// TwinCAT 3 PLC project PLC
// ProgramVersion: 3.1.4023.0
// libraries:
//   Tc2_Standard, * (Beckhoff Automation GmbH)
//   Tc2_System, * (Beckhoff Automation GmbH)
//   Tc3_Module, * (Beckhoff Automation GmbH)
// project tree:
//   / PlcTask.TcTTO
//   POUs/ MAIN.TcPOU
//   DUTs/IO/PdoEntries/ Status_E3F6A94B.TcDUT, Input_97D1F313.TcDUT, Status_B4798D86.TcDUT, Status_882A150F.TcDUT, Output_FFFF807A.TcDUT, Control_F189B737.TcDUT, Control_17BA1FC2.TcDUT
//   DUTs/IO/PDOs/ InfoData_6F19DB2B.TcDUT, Channel_42CA91F7.TcDUT, WcState_0B2B16F9.TcDUT, AI_Inputs_5AF6604E.TcDUT, WcState_9091E0EB.TcDUT, InfoData_32EB74EA.TcDUT, AI_Input_Channel_5AF6604E.TcDUT, Digital_BD004D6F.TcDUT, Encoder_Channel_2E4EA213.TcDUT, Digital_A7E1DFAB.TcDUT, Analog_Channel_5F9B7EA6.TcDUT, Encoder_Channel_B7999E14.TcDUT, DI_Inputs_BD004D6F.TcDUT, ENC_Inputs_Channel_69C51E8E.TcDUT, PLS_Inputs_5A35B63D.TcDUT, DO_Outputs_A7E1DFAB.TcDUT, AO_Output_Channel_BA7EBB7C.TcDUT, ENC_Outputs_Channel_DC4E290B.TcDUT, PLS_Outputs_AFB7DAF5.TcDUT, ENC_Inputs_Channel_6B6F9807.TcDUT, DI_Inputs_9882B618.TcDUT, ENC_Inputs_Channel_E5B5E929.TcDUT, PLS_Inputs_65C9A3D6.TcDUT, DO_Outputs_47E26D6A.TcDUT, ENC_Outputs_Channel_2E82BC43.TcDUT, PLS_Outputs_8EABC224.TcDUT, InfoData_E68C61CD.TcDUT, InfoData_2A97D6CF.TcDUT, Inputs_25A0042B.TcDUT, Outputs_2397A10E.TcDUT
//   DUTs/IO/Boxes/ EK1100_1FC0878B.TcDUT, EK1122_1FC0878B.TcDUT, EM2042_2B6483BD.TcDUT, EM3701_AB0D469D.TcDUT, EM3702_FDD84FD8.TcDUT, EM3712_FDD84FD8.TcDUT, EM7004_866015E1.TcDUT, EM7004_7586CC95.TcDUT, EM7004_5FA1DD22.TcDUT, EM7004_0F97553F.TcDUT
//   DUTs/IO/Devices/ SyncUnitTask_2D604ED5.TcDUT, SyncUnitTasks_6FEB8257.TcDUT, SyncUnits_99E584AF.TcDUT
//   DUTs/IO/Topology/ Beckhoff_EM2xxxEK1122_B7C04D41.TcDUT, Beckhoff_EM2xxx_23EB33C6.TcDUT, Beckhoff_EM3xxxEK1122_FEF78CCD.TcDUT, Beckhoff_EM3xxx_ABA31799.TcDUT, Beckhoff_EM7xxxEK1122_DEE9974A.TcDUT, Beckhoff_EM7xxx_9745B8AE.TcDUT, EtherCAT_Master_EMxxxx_E69B3047.TcDUT
//   DUTs/IO/Base/ EtcSlaveBase_82538BE2.TcDUT, EtcSlaveBase_82538BE2.TcDUT, EtcSlaveBase_82538BE2.TcDUT, EtcSlaveTerminalBase_947E5A46.TcDUT, EtcSlaveBoxBase_77A0E4A7.TcDUT, EtcSlaveEndTerminalBase_866C7F0C.TcDUT, InputBase_8311D824.TcDUT, OutputBase_10CEE7DE.TcDUT, EtcMasterBase_62654B43.TcDUT
//   GVLs/ GVL_iXlinker.TcGVL
// real-time tasks:
//   TASK PlcTask: cycle T#10ms, priority 20, ADS port 350
// I/O:
//   DEVICE EtherCAT_Master_EMxxxx, AmsNetId 172.20.30.238.12.1
//     Beckhoff EM2xxx [EK1100 EtherCAT Coupler (2A E-Bus)]
//       Beckhoff EM2xxxEK1122 [EK1122 2 port EtherCAT junction]
//         Beckhoff EM2xxxsub EK1100 [EK1100 EtherCAT Coupler (2A E-Bus)]
//       A_0001(EM2042-0000-0016) [EM2042 16Ch. Dig. Output 24V, 0.5A, D-Sub connection]
//       A_0002(EM2042-0000-0017) [EM2042 16Ch. Dig. Output 24V, 0.5A, D-Sub connection]
//     Beckhoff EM3xxx [EK1100 EtherCAT Coupler (2A E-Bus)]
//       Beckhoff EM3xxxEK1122 [EK1122 2 port EtherCAT junction]
//         Beckhoff EM3xxxsub EK1100 [EK1100 EtherCAT Coupler (2A E-Bus)]
//       A_0001(EM3701-0000-0016) [EM3701, 1Ch. differential pressure measuring terminal 100hPa (100mbar)]
//       A_0002(EM3702-0000-0016) [EM3702  2Ch. relative pressure measuring terminal 7,500 hPa (7.5 bar)]
//       A_0003(EM3712-0000-0016) [EM3712  2Ch relative pressure measuring terminal -1,000...+1,000 hPa (-1...+1 bar)]
//     Beckhoff EM7xxx [EK1100 EtherCAT Coupler (2A E-Bus)]
//       Beckhoff EM7xxxEK1122 [EK1122 2 port EtherCAT junction]
//         Beckhoff EM7xxxsub EK1100 [EK1100 EtherCAT Coupler (2A E-Bus)]
//       A_0001(EM7004-0000-9995) [EM7004 4-Axis Interface Unit]
//       A_0002(EM7004-0000-9996) [EM7004 4-Axis Interface Unit]
//       A_0003(EM7004-0000-9997) [EM7004 4-Axis Interface Unit]
//       A_0004(EM7004-0000-0016) [EM7004 4-Axis Interface Unit]
//       A_0005(EM7004-0000-0017) [EM7004 4-Axis Interface Unit]
//       A_0006(EM7004-0000-0018) [EM7004 4-Axis Interface Unit]
// variable links:
//   PLC/PLC Instance <-> EtherCAT Master EMxxxx/Beckhoff EM2xxx
//     PlcTask Inputs/GVL_iXlinker.EtherCAT_Master_EMxxxx.Beckhoff_EM2xxx.InfoData.State <-> InfoData/State
//   PLC/PLC Instance <-> EtherCAT Master EMxxxx/Beckhoff EM2xxx/Beckhoff EM2xxxEK1122
//     PlcTask Inputs/GVL_iXlinker.EtherCAT_Master_EMxxxx.Beckhoff_EM2xxx.Beckhoff_EM2xxxEK1122.InfoData.State <-> InfoData/State
//   PLC/PLC Instance <-> EtherCAT Master EMxxxx/Beckhoff EM2xxx/Beckhoff EM2xxxEK1122/Beckhoff EM2xxxsub EK1100
//     PlcTask Inputs/GVL_iXlinker.EtherCAT_Master_EMxxxx.Beckhoff_EM2xxx.Beckhoff_EM2xxxEK1122.Beckhoff_EM2xxxsub_EK1100.InfoData.State <-> InfoData/State
//   PLC/PLC Instance <-> EtherCAT Master EMxxxx/Beckhoff EM2xxx/A_0001(EM2042-0000-0016)
//     PlcTask Outputs/GVL_iXlinker.EtherCAT_Master_EMxxxx.Beckhoff_EM2xxx.A_0001_EM2042_0000_0016.Channel_1.Output <-> Channel 1/Output
//     PlcTask Outputs/GVL_iXlinker.EtherCAT_Master_EMxxxx.Beckhoff_EM2xxx.A_0001_EM2042_0000_0016.Channel_2.Output <-> Channel 2/Output
//     PlcTask Outputs/GVL_iXlinker.EtherCAT_Master_EMxxxx.Beckhoff_EM2xxx.A_0001_EM2042_0000_0016.Channel_3.Output <-> Channel 3/Output
//     PlcTask Outputs/GVL_iXlinker.EtherCAT_Master_EMxxxx.Beckhoff_EM2xxx.A_0001_EM2042_0000_0016.Channel_4.Output <-> Channel 4/Output
//     PlcTask Outputs/GVL_iXlinker.EtherCAT_Master_EMxxxx.Beckhoff_EM2xxx.A_0001_EM2042_0000_0016.Channel_5.Output <-> Channel 5/Output
//     PlcTask Outputs/GVL_iXlinker.EtherCAT_Master_EMxxxx.Beckhoff_EM2xxx.A_0001_EM2042_0000_0016.Channel_6.Output <-> Channel 6/Output
//     PlcTask Outputs/GVL_iXlinker.EtherCAT_Master_EMxxxx.Beckhoff_EM2xxx.A_0001_EM2042_0000_0016.Channel_7.Output <-> Channel 7/Output
//     PlcTask Outputs/GVL_iXlinker.EtherCAT_Master_EMxxxx.Beckhoff_EM2xxx.A_0001_EM2042_0000_0016.Channel_8.Output <-> Channel 8/Output
//     PlcTask Outputs/GVL_iXlinker.EtherCAT_Master_EMxxxx.Beckhoff_EM2xxx.A_0001_EM2042_0000_0016.Channel_9.Output <-> Channel 9/Output
//     PlcTask Outputs/GVL_iXlinker.EtherCAT_Master_EMxxxx.Beckhoff_EM2xxx.A_0001_EM2042_0000_0016.Channel_10.Output <-> Channel 10/Output
//     PlcTask Outputs/GVL_iXlinker.EtherCAT_Master_EMxxxx.Beckhoff_EM2xxx.A_0001_EM2042_0000_0016.Channel_11.Output <-> Channel 11/Output
//     PlcTask Outputs/GVL_iXlinker.EtherCAT_Master_EMxxxx.Beckhoff_EM2xxx.A_0001_EM2042_0000_0016.Channel_12.Output <-> Channel 12/Output
//     PlcTask Outputs/GVL_iXlinker.EtherCAT_Master_EMxxxx.Beckhoff_EM2xxx.A_0001_EM2042_0000_0016.Channel_13.Output <-> Channel 13/Output
//     PlcTask Outputs/GVL_iXlinker.EtherCAT_Master_EMxxxx.Beckhoff_EM2xxx.A_0001_EM2042_0000_0016.Channel_14.Output <-> Channel 14/Output
//     PlcTask Outputs/GVL_iXlinker.EtherCAT_Master_EMxxxx.Beckhoff_EM2xxx.A_0001_EM2042_0000_0016.Channel_15.Output <-> Channel 15/Output
//     PlcTask Outputs/GVL_iXlinker.EtherCAT_Master_EMxxxx.Beckhoff_EM2xxx.A_0001_EM2042_0000_0016.Channel_16.Output <-> Channel 16/Output
//     PlcTask Inputs/GVL_iXlinker.EtherCAT_Master_EMxxxx.Beckhoff_EM2xxx.A_0001_EM2042_0000_0016.WcState.WcState <-> WcState/WcState
//     PlcTask Inputs/GVL_iXlinker.EtherCAT_Master_EMxxxx.Beckhoff_EM2xxx.A_0001_EM2042_0000_0016.InfoData.State <-> InfoData/State
//   PLC/PLC Instance <-> EtherCAT Master EMxxxx/Beckhoff EM2xxx/A_0002(EM2042-0000-0017)
//     PlcTask Outputs/GVL_iXlinker.EtherCAT_Master_EMxxxx.Beckhoff_EM2xxx.A_0002_EM2042_0000_0017.Channel_1.Output <-> Channel 1/Output
//     PlcTask Outputs/GVL_iXlinker.EtherCAT_Master_EMxxxx.Beckhoff_EM2xxx.A_0002_EM2042_0000_0017.Channel_2.Output <-> Channel 2/Output
//     PlcTask Outputs/GVL_iXlinker.EtherCAT_Master_EMxxxx.Beckhoff_EM2xxx.A_0002_EM2042_0000_0017.Channel_3.Output <-> Channel 3/Output
//     PlcTask Outputs/GVL_iXlinker.EtherCAT_Master_EMxxxx.Beckhoff_EM2xxx.A_0002_EM2042_0000_0017.Channel_4.Output <-> Channel 4/Output
//     PlcTask Outputs/GVL_iXlinker.EtherCAT_Master_EMxxxx.Beckhoff_EM2xxx.A_0002_EM2042_0000_0017.Channel_5.Output <-> Channel 5/Output
//     PlcTask Outputs/GVL_iXlinker.EtherCAT_Master_EMxxxx.Beckhoff_EM2xxx.A_0002_EM2042_0000_0017.Channel_6.Output <-> Channel 6/Output
//     PlcTask Outputs/GVL_iXlinker.EtherCAT_Master_EMxxxx.Beckhoff_EM2xxx.A_0002_EM2042_0000_0017.Channel_7.Output <-> Channel 7/Output
//     PlcTask Outputs/GVL_iXlinker.EtherCAT_Master_EMxxxx.Beckhoff_EM2xxx.A_0002_EM2042_0000_0017.Channel_8.Output <-> Channel 8/Output
//     PlcTask Outputs/GVL_iXlinker.EtherCAT_Master_EMxxxx.Beckhoff_EM2xxx.A_0002_EM2042_0000_0017.Channel_9.Output <-> Channel 9/Output
//     PlcTask Outputs/GVL_iXlinker.EtherCAT_Master_EMxxxx.Beckhoff_EM2xxx.A_0002_EM2042_0000_0017.Channel_10.Output <-> Channel 10/Output
//     PlcTask Outputs/GVL_iXlinker.EtherCAT_Master_EMxxxx.Beckhoff_EM2xxx.A_0002_EM2042_0000_0017.Channel_11.Output <-> Channel 11/Output
//     PlcTask Outputs/GVL_iXlinker.EtherCAT_Master_EMxxxx.Beckhoff_EM2xxx.A_0002_EM2042_0000_0017.Channel_12.Output <-> Channel 12/Output
//     PlcTask Outputs/GVL_iXlinker.EtherCAT_Master_EMxxxx.Beckhoff_EM2xxx.A_0002_EM2042_0000_0017.Channel_13.Output <-> Channel 13/Output
//     PlcTask Outputs/GVL_iXlinker.EtherCAT_Master_EMxxxx.Beckhoff_EM2xxx.A_0002_EM2042_0000_0017.Channel_14.Output <-> Channel 14/Output
//     PlcTask Outputs/GVL_iXlinker.EtherCAT_Master_EMxxxx.Beckhoff_EM2xxx.A_0002_EM2042_0000_0017.Channel_15.Output <-> Channel 15/Output
//     PlcTask Outputs/GVL_iXlinker.EtherCAT_Master_EMxxxx.Beckhoff_EM2xxx.A_0002_EM2042_0000_0017.Channel_16.Output <-> Channel 16/Output
//     PlcTask Inputs/GVL_iXlinker.EtherCAT_Master_EMxxxx.Beckhoff_EM2xxx.A_0002_EM2042_0000_0017.WcState.WcState <-> WcState/WcState
//     PlcTask Inputs/GVL_iXlinker.EtherCAT_Master_EMxxxx.Beckhoff_EM2xxx.A_0002_EM2042_0000_0017.InfoData.State <-> InfoData/State
//   PLC/PLC Instance <-> EtherCAT Master EMxxxx/Beckhoff EM3xxx
//     PlcTask Inputs/GVL_iXlinker.EtherCAT_Master_EMxxxx.Beckhoff_EM3xxx.InfoData.State <-> InfoData/State
//   PLC/PLC Instance <-> EtherCAT Master EMxxxx/Beckhoff EM3xxx/Beckhoff EM3xxxEK1122
//     PlcTask Inputs/GVL_iXlinker.EtherCAT_Master_EMxxxx.Beckhoff_EM3xxx.Beckhoff_EM3xxxEK1122.InfoData.State <-> InfoData/State
//   PLC/PLC Instance <-> EtherCAT Master EMxxxx/Beckhoff EM3xxx/Beckhoff EM3xxxEK1122/Beckhoff EM3xxxsub EK1100
//     PlcTask Inputs/GVL_iXlinker.EtherCAT_Master_EMxxxx.Beckhoff_EM3xxx.Beckhoff_EM3xxxEK1122.Beckhoff_EM3xxxsub_EK1100.InfoData.State <-> InfoData/State
//   PLC/PLC Instance <-> EtherCAT Master EMxxxx/Beckhoff EM3xxx/A_0001(EM3701-0000-0016)
//     PlcTask Inputs/GVL_iXlinker.EtherCAT_Master_EMxxxx.Beckhoff_EM3xxx.A_0001_EM3701_0000_0016.AI_Inputs.Status/Underrange <-> AI Inputs/Status/Underrange
//     PlcTask Inputs/GVL_iXlinker.EtherCAT_Master_EMxxxx.Beckhoff_EM3xxx.A_0001_EM3701_0000_0016.AI_Inputs.Status/Overrange <-> AI Inputs/Status/Overrange
//     PlcTask Inputs/GVL_iXlinker.EtherCAT_Master_EMxxxx.Beckhoff_EM3xxx.A_0001_EM3701_0000_0016.AI_Inputs.Status/Limit_1 <-> AI Inputs/Status/Limit 1
//     PlcTask Inputs/GVL_iXlinker.EtherCAT_Master_EMxxxx.Beckhoff_EM3xxx.A_0001_EM3701_0000_0016.AI_Inputs.Status/Limit_2 <-> AI Inputs/Status/Limit 2
//     PlcTask Inputs/GVL_iXlinker.EtherCAT_Master_EMxxxx.Beckhoff_EM3xxx.A_0001_EM3701_0000_0016.AI_Inputs.Status/Error <-> AI Inputs/Status/Error
//     PlcTask Inputs/GVL_iXlinker.EtherCAT_Master_EMxxxx.Beckhoff_EM3xxx.A_0001_EM3701_0000_0016.AI_Inputs.Status/TxPDO_State <-> AI Inputs/Status/TxPDO State
//     PlcTask Inputs/GVL_iXlinker.EtherCAT_Master_EMxxxx.Beckhoff_EM3xxx.A_0001_EM3701_0000_0016.AI_Inputs.Value <-> AI Inputs/Value
//     PlcTask Inputs/GVL_iXlinker.EtherCAT_Master_EMxxxx.Beckhoff_EM3xxx.A_0001_EM3701_0000_0016.WcState.WcState <-> WcState/WcState
//     PlcTask Inputs/GVL_iXlinker.EtherCAT_Master_EMxxxx.Beckhoff_EM3xxx.A_0001_EM3701_0000_0016.WcState.InputToggle <-> WcState/InputToggle
//     PlcTask Inputs/GVL_iXlinker.EtherCAT_Master_EMxxxx.Beckhoff_EM3xxx.A_0001_EM3701_0000_0016.InfoData.AdsAddr <-> InfoData/AdsAddr
//     PlcTask Inputs/GVL_iXlinker.EtherCAT_Master_EMxxxx.Beckhoff_EM3xxx.A_0001_EM3701_0000_0016.InfoData.State <-> InfoData/State
//   PLC/PLC Instance <-> EtherCAT Master EMxxxx/Beckhoff EM3xxx/A_0002(EM3702-0000-0016)
//     PlcTask Inputs/GVL_iXlinker.EtherCAT_Master_EMxxxx.Beckhoff_EM3xxx.A_0002_EM3702_0000_0016.AI_Input_Channel_1.Status/Underrange <-> AI Input Channel 1/Status/Underrange
//     PlcTask Inputs/GVL_iXlinker.EtherCAT_Master_EMxxxx.Beckhoff_EM3xxx.A_0002_EM3702_0000_0016.AI_Input_Channel_2.Status/Underrange <-> AI Input Channel 2/Status/Underrange
//     PlcTask Inputs/GVL_iXlinker.EtherCAT_Master_EMxxxx.Beckhoff_EM3xxx.A_0002_EM3702_0000_0016.AI_Input_Channel_1.Status/Overrange <-> AI Input Channel 1/Status/Overrange
//     PlcTask Inputs/GVL_iXlinker.EtherCAT_Master_EMxxxx.Beckhoff_EM3xxx.A_0002_EM3702_0000_0016.AI_Input_Channel_2.Status/Overrange <-> AI Input Channel 2/Status/Overrange
//     PlcTask Inputs/GVL_iXlinker.EtherCAT_Master_EMxxxx.Beckhoff_EM3xxx.A_0002_EM3702_0000_0016.AI_Input_Channel_1.Status/Limit_1 <-> AI Input Channel 1/Status/Limit 1
//     PlcTask Inputs/GVL_iXlinker.EtherCAT_Master_EMxxxx.Beckhoff_EM3xxx.A_0002_EM3702_0000_0016.AI_Input_Channel_1.Status/Limit_2 <-> AI Input Channel 1/Status/Limit 2
//     PlcTask Inputs/GVL_iXlinker.EtherCAT_Master_EMxxxx.Beckhoff_EM3xxx.A_0002_EM3702_0000_0016.AI_Input_Channel_2.Status/Limit_1 <-> AI Input Channel 2/Status/Limit 1
//     PlcTask Inputs/GVL_iXlinker.EtherCAT_Master_EMxxxx.Beckhoff_EM3xxx.A_0002_EM3702_0000_0016.AI_Input_Channel_2.Status/Limit_2 <-> AI Input Channel 2/Status/Limit 2
//     PlcTask Inputs/GVL_iXlinker.EtherCAT_Master_EMxxxx.Beckhoff_EM3xxx.A_0002_EM3702_0000_0016.AI_Input_Channel_1.Status/Error <-> AI Input Channel 1/Status/Error
//     PlcTask Inputs/GVL_iXlinker.EtherCAT_Master_EMxxxx.Beckhoff_EM3xxx.A_0002_EM3702_0000_0016.AI_Input_Channel_2.Status/Error <-> AI Input Channel 2/Status/Error
//     PlcTask Inputs/GVL_iXlinker.EtherCAT_Master_EMxxxx.Beckhoff_EM3xxx.A_0002_EM3702_0000_0016.AI_Input_Channel_1.Status/TxPDO_State <-> AI Input Channel 1/Status/TxPDO State
//     PlcTask Inputs/GVL_iXlinker.EtherCAT_Master_EMxxxx.Beckhoff_EM3xxx.A_0002_EM3702_0000_0016.AI_Input_Channel_2.Status/TxPDO_State <-> AI Input Channel 2/Status/TxPDO State
//     PlcTask Inputs/GVL_iXlinker.EtherCAT_Master_EMxxxx.Beckhoff_EM3xxx.A_0002_EM3702_0000_0016.AI_Input_Channel_1.Value <-> AI Input Channel 1/Value
//     PlcTask Inputs/GVL_iXlinker.EtherCAT_Master_EMxxxx.Beckhoff_EM3xxx.A_0002_EM3702_0000_0016.AI_Input_Channel_2.Value <-> AI Input Channel 2/Value
//     PlcTask Inputs/GVL_iXlinker.EtherCAT_Master_EMxxxx.Beckhoff_EM3xxx.A_0002_EM3702_0000_0016.WcState.WcState <-> WcState/WcState
//     PlcTask Inputs/GVL_iXlinker.EtherCAT_Master_EMxxxx.Beckhoff_EM3xxx.A_0002_EM3702_0000_0016.WcState.InputToggle <-> WcState/InputToggle
//     PlcTask Inputs/GVL_iXlinker.EtherCAT_Master_EMxxxx.Beckhoff_EM3xxx.A_0002_EM3702_0000_0016.InfoData.AdsAddr <-> InfoData/AdsAddr
//     PlcTask Inputs/GVL_iXlinker.EtherCAT_Master_EMxxxx.Beckhoff_EM3xxx.A_0002_EM3702_0000_0016.InfoData.State <-> InfoData/State
//   PLC/PLC Instance <-> EtherCAT Master EMxxxx/Beckhoff EM3xxx/A_0003(EM3712-0000-0016)
//     PlcTask Inputs/GVL_iXlinker.EtherCAT_Master_EMxxxx.Beckhoff_EM3xxx.A_0003_EM3712_0000_0016.AI_Input_Channel_1.Status/Underrange <-> AI Input Channel 1/Status/Underrange
//     PlcTask Inputs/GVL_iXlinker.EtherCAT_Master_EMxxxx.Beckhoff_EM3xxx.A_0003_EM3712_0000_0016.AI_Input_Channel_2.Status/Underrange <-> AI Input Channel 2/Status/Underrange
//     PlcTask Inputs/GVL_iXlinker.EtherCAT_Master_EMxxxx.Beckhoff_EM3xxx.A_0003_EM3712_0000_0016.AI_Input_Channel_1.Status/Overrange <-> AI Input Channel 1/Status/Overrange
//     PlcTask Inputs/GVL_iXlinker.EtherCAT_Master_EMxxxx.Beckhoff_EM3xxx.A_0003_EM3712_0000_0016.AI_Input_Channel_2.Status/Overrange <-> AI Input Channel 2/Status/Overrange
//     PlcTask Inputs/GVL_iXlinker.EtherCAT_Master_EMxxxx.Beckhoff_EM3xxx.A_0003_EM3712_0000_0016.AI_Input_Channel_1.Status/Limit_1 <-> AI Input Channel 1/Status/Limit 1
//     PlcTask Inputs/GVL_iXlinker.EtherCAT_Master_EMxxxx.Beckhoff_EM3xxx.A_0003_EM3712_0000_0016.AI_Input_Channel_1.Status/Limit_2 <-> AI Input Channel 1/Status/Limit 2
//     PlcTask Inputs/GVL_iXlinker.EtherCAT_Master_EMxxxx.Beckhoff_EM3xxx.A_0003_EM3712_0000_0016.AI_Input_Channel_2.Status/Limit_1 <-> AI Input Channel 2/Status/Limit 1
//     PlcTask Inputs/GVL_iXlinker.EtherCAT_Master_EMxxxx.Beckhoff_EM3xxx.A_0003_EM3712_0000_0016.AI_Input_Channel_2.Status/Limit_2 <-> AI Input Channel 2/Status/Limit 2
//     PlcTask Inputs/GVL_iXlinker.EtherCAT_Master_EMxxxx.Beckhoff_EM3xxx.A_0003_EM3712_0000_0016.AI_Input_Channel_1.Status/Error <-> AI Input Channel 1/Status/Error
//     PlcTask Inputs/GVL_iXlinker.EtherCAT_Master_EMxxxx.Beckhoff_EM3xxx.A_0003_EM3712_0000_0016.AI_Input_Channel_2.Status/Error <-> AI Input Channel 2/Status/Error
//     PlcTask Inputs/GVL_iXlinker.EtherCAT_Master_EMxxxx.Beckhoff_EM3xxx.A_0003_EM3712_0000_0016.AI_Input_Channel_1.Status/TxPDO_State <-> AI Input Channel 1/Status/TxPDO State
//     PlcTask Inputs/GVL_iXlinker.EtherCAT_Master_EMxxxx.Beckhoff_EM3xxx.A_0003_EM3712_0000_0016.AI_Input_Channel_2.Status/TxPDO_State <-> AI Input Channel 2/Status/TxPDO State
//     PlcTask Inputs/GVL_iXlinker.EtherCAT_Master_EMxxxx.Beckhoff_EM3xxx.A_0003_EM3712_0000_0016.AI_Input_Channel_1.Value <-> AI Input Channel 1/Value
//     PlcTask Inputs/GVL_iXlinker.EtherCAT_Master_EMxxxx.Beckhoff_EM3xxx.A_0003_EM3712_0000_0016.AI_Input_Channel_2.Value <-> AI Input Channel 2/Value
//     PlcTask Inputs/GVL_iXlinker.EtherCAT_Master_EMxxxx.Beckhoff_EM3xxx.A_0003_EM3712_0000_0016.WcState.WcState <-> WcState/WcState
//     PlcTask Inputs/GVL_iXlinker.EtherCAT_Master_EMxxxx.Beckhoff_EM3xxx.A_0003_EM3712_0000_0016.WcState.InputToggle <-> WcState/InputToggle
//     PlcTask Inputs/GVL_iXlinker.EtherCAT_Master_EMxxxx.Beckhoff_EM3xxx.A_0003_EM3712_0000_0016.InfoData.AdsAddr <-> InfoData/AdsAddr
//     PlcTask Inputs/GVL_iXlinker.EtherCAT_Master_EMxxxx.Beckhoff_EM3xxx.A_0003_EM3712_0000_0016.InfoData.State <-> InfoData/State
//   PLC/PLC Instance <-> EtherCAT Master EMxxxx/Beckhoff EM7xxx
//     PlcTask Inputs/GVL_iXlinker.EtherCAT_Master_EMxxxx.Beckhoff_EM7xxx.InfoData.State <-> InfoData/State
//   PLC/PLC Instance <-> EtherCAT Master EMxxxx/Beckhoff EM7xxx/Beckhoff EM7xxxEK1122
//     PlcTask Inputs/GVL_iXlinker.EtherCAT_Master_EMxxxx.Beckhoff_EM7xxx.Beckhoff_EM7xxxEK1122.InfoData.State <-> InfoData/State
//   PLC/PLC Instance <-> EtherCAT Master EMxxxx/Beckhoff EM7xxx/Beckhoff EM7xxxEK1122/Beckhoff EM7xxxsub EK1100
//     PlcTask Inputs/GVL_iXlinker.EtherCAT_Master_EMxxxx.Beckhoff_EM7xxx.Beckhoff_EM7xxxEK1122.Beckhoff_EM7xxxsub_EK1100.InfoData.State <-> InfoData/State
//   PLC/PLC Instance <-> EtherCAT Master EMxxxx/Beckhoff EM7xxx/A_0001(EM7004-0000-9995)
//     PlcTask Inputs/GVL_iXlinker.EtherCAT_Master_EMxxxx.Beckhoff_EM7xxx.A_0001_EM7004_0000_9995.Digital.Input[0] <-> Digital/Input 0
//     PlcTask Inputs/GVL_iXlinker.EtherCAT_Master_EMxxxx.Beckhoff_EM7xxx.A_0001_EM7004_0000_9995.Digital.Input[1] <-> Digital/Input 1
//     PlcTask Inputs/GVL_iXlinker.EtherCAT_Master_EMxxxx.Beckhoff_EM7xxx.A_0001_EM7004_0000_9995.Digital.Input[2] <-> Digital/Input 2
//     PlcTask Inputs/GVL_iXlinker.EtherCAT_Master_EMxxxx.Beckhoff_EM7xxx.A_0001_EM7004_0000_9995.Digital.Input[3] <-> Digital/Input 3
//     PlcTask Inputs/GVL_iXlinker.EtherCAT_Master_EMxxxx.Beckhoff_EM7xxx.A_0001_EM7004_0000_9995.Digital.Input[4] <-> Digital/Input 4
//     PlcTask Inputs/GVL_iXlinker.EtherCAT_Master_EMxxxx.Beckhoff_EM7xxx.A_0001_EM7004_0000_9995.Digital.Input[5] <-> Digital/Input 5
//     PlcTask Inputs/GVL_iXlinker.EtherCAT_Master_EMxxxx.Beckhoff_EM7xxx.A_0001_EM7004_0000_9995.Digital.Input[6] <-> Digital/Input 6
//     PlcTask Inputs/GVL_iXlinker.EtherCAT_Master_EMxxxx.Beckhoff_EM7xxx.A_0001_EM7004_0000_9995.Digital.Input[7] <-> Digital/Input 7
//     PlcTask Inputs/GVL_iXlinker.EtherCAT_Master_EMxxxx.Beckhoff_EM7xxx.A_0001_EM7004_0000_9995.Digital.Input[8] <-> Digital/Input 8
//     PlcTask Inputs/GVL_iXlinker.EtherCAT_Master_EMxxxx.Beckhoff_EM7xxx.A_0001_EM7004_0000_9995.Digital.Input[9] <-> Digital/Input 9
//     PlcTask Inputs/GVL_iXlinker.EtherCAT_Master_EMxxxx.Beckhoff_EM7xxx.A_0001_EM7004_0000_9995.Digital.Input[10] <-> Digital/Input 10
//     PlcTask Inputs/GVL_iXlinker.EtherCAT_Master_EMxxxx.Beckhoff_EM7xxx.A_0001_EM7004_0000_9995.Digital.Input[11] <-> Digital/Input 11
//     PlcTask Inputs/GVL_iXlinker.EtherCAT_Master_EMxxxx.Beckhoff_EM7xxx.A_0001_EM7004_0000_9995.Digital.Input[12] <-> Digital/Input 12
//     PlcTask Inputs/GVL_iXlinker.EtherCAT_Master_EMxxxx.Beckhoff_EM7xxx.A_0001_EM7004_0000_9995.Digital.Input[13] <-> Digital/Input 13
//     PlcTask Inputs/GVL_iXlinker.EtherCAT_Master_EMxxxx.Beckhoff_EM7xxx.A_0001_EM7004_0000_9995.Digital.Input[14] <-> Digital/Input 14
//     PlcTask Inputs/GVL_iXlinker.EtherCAT_Master_EMxxxx.Beckhoff_EM7xxx.A_0001_EM7004_0000_9995.Digital.Input[15] <-> Digital/Input 15
//     PlcTask Inputs/GVL_iXlinker.EtherCAT_Master_EMxxxx.Beckhoff_EM7xxx.A_0001_EM7004_0000_9995.Encoder_Channel_1.Status <-> Encoder, Channel 1/Status
//     PlcTask Inputs/GVL_iXlinker.EtherCAT_Master_EMxxxx.Beckhoff_EM7xxx.A_0001_EM7004_0000_9995.Encoder_Channel_2.Status <-> Encoder, Channel 2/Status
//     PlcTask Inputs/GVL_iXlinker.EtherCAT_Master_EMxxxx.Beckhoff_EM7xxx.A_0001_EM7004_0000_9995.Encoder_Channel_3.Status <-> Encoder, Channel 3/Status
//     PlcTask Inputs/GVL_iXlinker.EtherCAT_Master_EMxxxx.Beckhoff_EM7xxx.A_0001_EM7004_0000_9995.Encoder_Channel_4.Status <-> Encoder, Channel 4/Status
//     PlcTask Inputs/GVL_iXlinker.EtherCAT_Master_EMxxxx.Beckhoff_EM7xxx.A_0001_EM7004_0000_9995.Encoder_Channel_1.Value <-> Encoder, Channel 1/Value
//     PlcTask Inputs/GVL_iXlinker.EtherCAT_Master_EMxxxx.Beckhoff_EM7xxx.A_0001_EM7004_0000_9995.Encoder_Channel_2.Value <-> Encoder, Channel 2/Value
//     PlcTask Inputs/GVL_iXlinker.EtherCAT_Master_EMxxxx.Beckhoff_EM7xxx.A_0001_EM7004_0000_9995.Encoder_Channel_3.Value <-> Encoder, Channel 3/Value
//     PlcTask Inputs/GVL_iXlinker.EtherCAT_Master_EMxxxx.Beckhoff_EM7xxx.A_0001_EM7004_0000_9995.Encoder_Channel_4.Value <-> Encoder, Channel 4/Value
//     PlcTask Inputs/GVL_iXlinker.EtherCAT_Master_EMxxxx.Beckhoff_EM7xxx.A_0001_EM7004_0000_9995.Encoder_Channel_1.Latch <-> Encoder, Channel 1/Latch
//     PlcTask Inputs/GVL_iXlinker.EtherCAT_Master_EMxxxx.Beckhoff_EM7xxx.A_0001_EM7004_0000_9995.Encoder_Channel_2.Latch <-> Encoder, Channel 2/Latch
//     PlcTask Inputs/GVL_iXlinker.EtherCAT_Master_EMxxxx.Beckhoff_EM7xxx.A_0001_EM7004_0000_9995.Encoder_Channel_3.Latch <-> Encoder, Channel 3/Latch
//     PlcTask Inputs/GVL_iXlinker.EtherCAT_Master_EMxxxx.Beckhoff_EM7xxx.A_0001_EM7004_0000_9995.Encoder_Channel_4.Latch <-> Encoder, Channel 4/Latch
//     PlcTask Outputs/GVL_iXlinker.EtherCAT_Master_EMxxxx.Beckhoff_EM7xxx.A_0001_EM7004_0000_9995.Digital_1.Output[0] <-> Digital_1/Output 0
//     PlcTask Outputs/GVL_iXlinker.EtherCAT_Master_EMxxxx.Beckhoff_EM7xxx.A_0001_EM7004_0000_9995.Digital_1.Output[1] <-> Digital_1/Output 1
//     PlcTask Outputs/GVL_iXlinker.EtherCAT_Master_EMxxxx.Beckhoff_EM7xxx.A_0001_EM7004_0000_9995.Digital_1.Output[2] <-> Digital_1/Output 2
//     PlcTask Outputs/GVL_iXlinker.EtherCAT_Master_EMxxxx.Beckhoff_EM7xxx.A_0001_EM7004_0000_9995.Digital_1.Output[3] <-> Digital_1/Output 3
//     PlcTask Outputs/GVL_iXlinker.EtherCAT_Master_EMxxxx.Beckhoff_EM7xxx.A_0001_EM7004_0000_9995.Digital_1.Output[4] <-> Digital_1/Output 4
//     PlcTask Outputs/GVL_iXlinker.EtherCAT_Master_EMxxxx.Beckhoff_EM7xxx.A_0001_EM7004_0000_9995.Digital_1.Output[5] <-> Digital_1/Output 5
//     PlcTask Outputs/GVL_iXlinker.EtherCAT_Master_EMxxxx.Beckhoff_EM7xxx.A_0001_EM7004_0000_9995.Digital_1.Output[6] <-> Digital_1/Output 6
//     PlcTask Outputs/GVL_iXlinker.EtherCAT_Master_EMxxxx.Beckhoff_EM7xxx.A_0001_EM7004_0000_9995.Digital_1.Output[7] <-> Digital_1/Output 7
//     PlcTask Outputs/GVL_iXlinker.EtherCAT_Master_EMxxxx.Beckhoff_EM7xxx.A_0001_EM7004_0000_9995.Digital_1.Output[8] <-> Digital_1/Output 8
//     PlcTask Outputs/GVL_iXlinker.EtherCAT_Master_EMxxxx.Beckhoff_EM7xxx.A_0001_EM7004_0000_9995.Digital_1.Output[9] <-> Digital_1/Output 9
//     PlcTask Outputs/GVL_iXlinker.EtherCAT_Master_EMxxxx.Beckhoff_EM7xxx.A_0001_EM7004_0000_9995.Digital_1.Output[10] <-> Digital_1/Output 10
//     PlcTask Outputs/GVL_iXlinker.EtherCAT_Master_EMxxxx.Beckhoff_EM7xxx.A_0001_EM7004_0000_9995.Digital_1.Output[11] <-> Digital_1/Output 11
//     PlcTask Outputs/GVL_iXlinker.EtherCAT_Master_EMxxxx.Beckhoff_EM7xxx.A_0001_EM7004_0000_9995.Digital_1.Output[12] <-> Digital_1/Output 12
//     PlcTask Outputs/GVL_iXlinker.EtherCAT_Master_EMxxxx.Beckhoff_EM7xxx.A_0001_EM7004_0000_9995.Digital_1.Output[13] <-> Digital_1/Output 13
//     PlcTask Outputs/GVL_iXlinker.EtherCAT_Master_EMxxxx.Beckhoff_EM7xxx.A_0001_EM7004_0000_9995.Digital_1.Output[14] <-> Digital_1/Output 14
//     PlcTask Outputs/GVL_iXlinker.EtherCAT_Master_EMxxxx.Beckhoff_EM7xxx.A_0001_EM7004_0000_9995.Digital_1.Output[15] <-> Digital_1/Output 15
//     PlcTask Outputs/GVL_iXlinker.EtherCAT_Master_EMxxxx.Beckhoff_EM7xxx.A_0001_EM7004_0000_9995.Analog_Channel_1.Output <-> Analog, Channel 1/Output
//     PlcTask Outputs/GVL_iXlinker.EtherCAT_Master_EMxxxx.Beckhoff_EM7xxx.A_0001_EM7004_0000_9995.Analog_Channel_2.Output <-> Analog, Channel 2/Output
//     PlcTask Outputs/GVL_iXlinker.EtherCAT_Master_EMxxxx.Beckhoff_EM7xxx.A_0001_EM7004_0000_9995.Analog_Channel_3.Output <-> Analog, Channel 3/Output
//     PlcTask Outputs/GVL_iXlinker.EtherCAT_Master_EMxxxx.Beckhoff_EM7xxx.A_0001_EM7004_0000_9995.Analog_Channel_4.Output <-> Analog, Channel 4/Output
//     PlcTask Outputs/GVL_iXlinker.EtherCAT_Master_EMxxxx.Beckhoff_EM7xxx.A_0001_EM7004_0000_9995.Encoder_Channel_1_1.Ctrl <-> Encoder, Channel 1_1/Ctrl
//     PlcTask Outputs/GVL_iXlinker.EtherCAT_Master_EMxxxx.Beckhoff_EM7xxx.A_0001_EM7004_0000_9995.Encoder_Channel_2_1.Ctrl <-> Encoder, Channel 2_1/Ctrl
//     PlcTask Outputs/GVL_iXlinker.EtherCAT_Master_EMxxxx.Beckhoff_EM7xxx.A_0001_EM7004_0000_9995.Encoder_Channel_3_1.Ctrl <-> Encoder, Channel 3_1/Ctrl
//     PlcTask Outputs/GVL_iXlinker.EtherCAT_Master_EMxxxx.Beckhoff_EM7xxx.A_0001_EM7004_0000_9995.Encoder_Channel_4_1.Ctrl <-> Encoder, Channel 4_1/Ctrl
//     PlcTask Outputs/GVL_iXlinker.EtherCAT_Master_EMxxxx.Beckhoff_EM7xxx.A_0001_EM7004_0000_9995.Encoder_Channel_1_1.Value <-> Encoder, Channel 1_1/Value
//     PlcTask Outputs/GVL_iXlinker.EtherCAT_Master_EMxxxx.Beckhoff_EM7xxx.A_0001_EM7004_0000_9995.Encoder_Channel_2_1.Value <-> Encoder, Channel 2_1/Value
//     PlcTask Outputs/GVL_iXlinker.EtherCAT_Master_EMxxxx.Beckhoff_EM7xxx.A_0001_EM7004_0000_9995.Encoder_Channel_3_1.Value <-> Encoder, Channel 3_1/Value
//     PlcTask Outputs/GVL_iXlinker.EtherCAT_Master_EMxxxx.Beckhoff_EM7xxx.A_0001_EM7004_0000_9995.Encoder_Channel_4_1.Value <-> Encoder, Channel 4_1/Value
//     PlcTask Inputs/GVL_iXlinker.EtherCAT_Master_EMxxxx.Beckhoff_EM7xxx.A_0001_EM7004_0000_9995.WcState.WcState <-> WcState/WcState
//     PlcTask Inputs/GVL_iXlinker.EtherCAT_Master_EMxxxx.Beckhoff_EM7xxx.A_0001_EM7004_0000_9995.WcState.InputToggle <-> WcState/InputToggle
//     PlcTask Inputs/GVL_iXlinker.EtherCAT_Master_EMxxxx.Beckhoff_EM7xxx.A_0001_EM7004_0000_9995.InfoData.AdsAddr <-> InfoData/AdsAddr
//     PlcTask Inputs/GVL_iXlinker.EtherCAT_Master_EMxxxx.Beckhoff_EM7xxx.A_0001_EM7004_0000_9995.InfoData.State <-> InfoData/State
//   PLC/PLC Instance <-> EtherCAT Master EMxxxx/Beckhoff EM7xxx/A_0002(EM7004-0000-9996)
//     PlcTask Inputs/GVL_iXlinker.EtherCAT_Master_EMxxxx.Beckhoff_EM7xxx.A_0002_EM7004_0000_9996.DI_Inputs.Input[0] <-> DI Inputs/Input 0
//     PlcTask Inputs/GVL_iXlinker.EtherCAT_Master_EMxxxx.Beckhoff_EM7xxx.A_0002_EM7004_0000_9996.DI_Inputs.Input[1] <-> DI Inputs/Input 1
//     PlcTask Inputs/GVL_iXlinker.EtherCAT_Master_EMxxxx.Beckhoff_EM7xxx.A_0002_EM7004_0000_9996.DI_Inputs.Input[2] <-> DI Inputs/Input 2
//     PlcTask Inputs/GVL_iXlinker.EtherCAT_Master_EMxxxx.Beckhoff_EM7xxx.A_0002_EM7004_0000_9996.DI_Inputs.Input[3] <-> DI Inputs/Input 3
//     PlcTask Inputs/GVL_iXlinker.EtherCAT_Master_EMxxxx.Beckhoff_EM7xxx.A_0002_EM7004_0000_9996.DI_Inputs.Input[4] <-> DI Inputs/Input 4
//     PlcTask Inputs/GVL_iXlinker.EtherCAT_Master_EMxxxx.Beckhoff_EM7xxx.A_0002_EM7004_0000_9996.DI_Inputs.Input[5] <-> DI Inputs/Input 5
//     PlcTask Inputs/GVL_iXlinker.EtherCAT_Master_EMxxxx.Beckhoff_EM7xxx.A_0002_EM7004_0000_9996.DI_Inputs.Input[6] <-> DI Inputs/Input 6
//     PlcTask Inputs/GVL_iXlinker.EtherCAT_Master_EMxxxx.Beckhoff_EM7xxx.A_0002_EM7004_0000_9996.DI_Inputs.Input[7] <-> DI Inputs/Input 7
//     PlcTask Inputs/GVL_iXlinker.EtherCAT_Master_EMxxxx.Beckhoff_EM7xxx.A_0002_EM7004_0000_9996.DI_Inputs.Input[8] <-> DI Inputs/Input 8
//     PlcTask Inputs/GVL_iXlinker.EtherCAT_Master_EMxxxx.Beckhoff_EM7xxx.A_0002_EM7004_0000_9996.DI_Inputs.Input[9] <-> DI Inputs/Input 9
//     PlcTask Inputs/GVL_iXlinker.EtherCAT_Master_EMxxxx.Beckhoff_EM7xxx.A_0002_EM7004_0000_9996.DI_Inputs.Input[10] <-> DI Inputs/Input 10
//     PlcTask Inputs/GVL_iXlinker.EtherCAT_Master_EMxxxx.Beckhoff_EM7xxx.A_0002_EM7004_0000_9996.DI_Inputs.Input[11] <-> DI Inputs/Input 11
//     PlcTask Inputs/GVL_iXlinker.EtherCAT_Master_EMxxxx.Beckhoff_EM7xxx.A_0002_EM7004_0000_9996.DI_Inputs.Input[12] <-> DI Inputs/Input 12
//     PlcTask Inputs/GVL_iXlinker.EtherCAT_Master_EMxxxx.Beckhoff_EM7xxx.A_0002_EM7004_0000_9996.DI_Inputs.Input[13] <-> DI Inputs/Input 13
//     PlcTask Inputs/GVL_iXlinker.EtherCAT_Master_EMxxxx.Beckhoff_EM7xxx.A_0002_EM7004_0000_9996.DI_Inputs.Input[14] <-> DI Inputs/Input 14
//     PlcTask Inputs/GVL_iXlinker.EtherCAT_Master_EMxxxx.Beckhoff_EM7xxx.A_0002_EM7004_0000_9996.DI_Inputs.Input[15] <-> DI Inputs/Input 15
//     PlcTask Inputs/GVL_iXlinker.EtherCAT_Master_EMxxxx.Beckhoff_EM7xxx.A_0002_EM7004_0000_9996.ENC_Inputs_Channel_1.Latch_extern_valid <-> ENC Inputs Channel 1/Latch extern valid
//     PlcTask Inputs/GVL_iXlinker.EtherCAT_Master_EMxxxx.Beckhoff_EM7xxx.A_0002_EM7004_0000_9996.ENC_Inputs_Channel_2.Latch_extern_valid <-> ENC Inputs Channel 2/Latch extern valid
//     PlcTask Inputs/GVL_iXlinker.EtherCAT_Master_EMxxxx.Beckhoff_EM7xxx.A_0002_EM7004_0000_9996.ENC_Inputs_Channel_3.Latch_extern_valid <-> ENC Inputs Channel 3/Latch extern valid
//     PlcTask Inputs/GVL_iXlinker.EtherCAT_Master_EMxxxx.Beckhoff_EM7xxx.A_0002_EM7004_0000_9996.ENC_Inputs_Channel_4.Latch_extern_valid <-> ENC Inputs Channel 4/Latch extern valid
//     PlcTask Inputs/GVL_iXlinker.EtherCAT_Master_EMxxxx.Beckhoff_EM7xxx.A_0002_EM7004_0000_9996.ENC_Inputs_Channel_1.Set_counter_done <-> ENC Inputs Channel 1/Set counter done
//     PlcTask Inputs/GVL_iXlinker.EtherCAT_Master_EMxxxx.Beckhoff_EM7xxx.A_0002_EM7004_0000_9996.ENC_Inputs_Channel_2.Set_counter_done <-> ENC Inputs Channel 2/Set counter done
//     PlcTask Inputs/GVL_iXlinker.EtherCAT_Master_EMxxxx.Beckhoff_EM7xxx.A_0002_EM7004_0000_9996.ENC_Inputs_Channel_3.Set_counter_done <-> ENC Inputs Channel 3/Set counter done
//     PlcTask Inputs/GVL_iXlinker.EtherCAT_Master_EMxxxx.Beckhoff_EM7xxx.A_0002_EM7004_0000_9996.ENC_Inputs_Channel_4.Set_counter_done <-> ENC Inputs Channel 4/Set counter done
//     PlcTask Inputs/GVL_iXlinker.EtherCAT_Master_EMxxxx.Beckhoff_EM7xxx.A_0002_EM7004_0000_9996.ENC_Inputs_Channel_1.Status_of_input_A <-> ENC Inputs Channel 1/Status of input A
//     PlcTask Inputs/GVL_iXlinker.EtherCAT_Master_EMxxxx.Beckhoff_EM7xxx.A_0002_EM7004_0000_9996.ENC_Inputs_Channel_2.Status_of_input_A <-> ENC Inputs Channel 2/Status of input A
//     PlcTask Inputs/GVL_iXlinker.EtherCAT_Master_EMxxxx.Beckhoff_EM7xxx.A_0002_EM7004_0000_9996.ENC_Inputs_Channel_3.Status_of_input_A <-> ENC Inputs Channel 3/Status of input A
//     PlcTask Inputs/GVL_iXlinker.EtherCAT_Master_EMxxxx.Beckhoff_EM7xxx.A_0002_EM7004_0000_9996.ENC_Inputs_Channel_4.Status_of_input_A <-> ENC Inputs Channel 4/Status of input A
//     PlcTask Inputs/GVL_iXlinker.EtherCAT_Master_EMxxxx.Beckhoff_EM7xxx.A_0002_EM7004_0000_9996.ENC_Inputs_Channel_1.Status_of_input_B <-> ENC Inputs Channel 1/Status of input B
//     PlcTask Inputs/GVL_iXlinker.EtherCAT_Master_EMxxxx.Beckhoff_EM7xxx.A_0002_EM7004_0000_9996.ENC_Inputs_Channel_2.Status_of_input_B <-> ENC Inputs Channel 2/Status of input B
//     PlcTask Inputs/GVL_iXlinker.EtherCAT_Master_EMxxxx.Beckhoff_EM7xxx.A_0002_EM7004_0000_9996.ENC_Inputs_Channel_3.Status_of_input_B <-> ENC Inputs Channel 3/Status of input B
//     PlcTask Inputs/GVL_iXlinker.EtherCAT_Master_EMxxxx.Beckhoff_EM7xxx.A_0002_EM7004_0000_9996.ENC_Inputs_Channel_4.Status_of_input_B <-> ENC Inputs Channel 4/Status of input B
//     PlcTask Inputs/GVL_iXlinker.EtherCAT_Master_EMxxxx.Beckhoff_EM7xxx.A_0002_EM7004_0000_9996.ENC_Inputs_Channel_1.Status_of_input_gate <-> ENC Inputs Channel 1/Status of input gate
//     PlcTask Inputs/GVL_iXlinker.EtherCAT_Master_EMxxxx.Beckhoff_EM7xxx.A_0002_EM7004_0000_9996.ENC_Inputs_Channel_2.Status_of_input_gate <-> ENC Inputs Channel 2/Status of input gate
//     PlcTask Inputs/GVL_iXlinker.EtherCAT_Master_EMxxxx.Beckhoff_EM7xxx.A_0002_EM7004_0000_9996.ENC_Inputs_Channel_3.Status_of_input_gate <-> ENC Inputs Channel 3/Status of input gate
//     PlcTask Inputs/GVL_iXlinker.EtherCAT_Master_EMxxxx.Beckhoff_EM7xxx.A_0002_EM7004_0000_9996.ENC_Inputs_Channel_4.Status_of_input_gate <-> ENC Inputs Channel 4/Status of input gate
//     PlcTask Inputs/GVL_iXlinker.EtherCAT_Master_EMxxxx.Beckhoff_EM7xxx.A_0002_EM7004_0000_9996.ENC_Inputs_Channel_1.Status_of_extern_latch <-> ENC Inputs Channel 1/Status of extern latch
//     PlcTask Inputs/GVL_iXlinker.EtherCAT_Master_EMxxxx.Beckhoff_EM7xxx.A_0002_EM7004_0000_9996.ENC_Inputs_Channel_2.Status_of_extern_latch <-> ENC Inputs Channel 2/Status of extern latch
//     PlcTask Inputs/GVL_iXlinker.EtherCAT_Master_EMxxxx.Beckhoff_EM7xxx.A_0002_EM7004_0000_9996.ENC_Inputs_Channel_3.Status_of_extern_latch <-> ENC Inputs Channel 3/Status of extern latch
//     PlcTask Inputs/GVL_iXlinker.EtherCAT_Master_EMxxxx.Beckhoff_EM7xxx.A_0002_EM7004_0000_9996.ENC_Inputs_Channel_4.Status_of_extern_latch <-> ENC Inputs Channel 4/Status of extern latch
//     PlcTask Inputs/GVL_iXlinker.EtherCAT_Master_EMxxxx.Beckhoff_EM7xxx.A_0002_EM7004_0000_9996.ENC_Inputs_Channel_1.Counter_value <-> ENC Inputs Channel 1/Counter value
//     PlcTask Inputs/GVL_iXlinker.EtherCAT_Master_EMxxxx.Beckhoff_EM7xxx.A_0002_EM7004_0000_9996.ENC_Inputs_Channel_2.Counter_value <-> ENC Inputs Channel 2/Counter value
//     PlcTask Inputs/GVL_iXlinker.EtherCAT_Master_EMxxxx.Beckhoff_EM7xxx.A_0002_EM7004_0000_9996.ENC_Inputs_Channel_3.Counter_value <-> ENC Inputs Channel 3/Counter value
//     PlcTask Inputs/GVL_iXlinker.EtherCAT_Master_EMxxxx.Beckhoff_EM7xxx.A_0002_EM7004_0000_9996.ENC_Inputs_Channel_4.Counter_value <-> ENC Inputs Channel 4/Counter value
//     PlcTask Inputs/GVL_iXlinker.EtherCAT_Master_EMxxxx.Beckhoff_EM7xxx.A_0002_EM7004_0000_9996.ENC_Inputs_Channel_1.Latch_value <-> ENC Inputs Channel 1/Latch value
//     PlcTask Inputs/GVL_iXlinker.EtherCAT_Master_EMxxxx.Beckhoff_EM7xxx.A_0002_EM7004_0000_9996.ENC_Inputs_Channel_2.Latch_value <-> ENC Inputs Channel 2/Latch value
//     PlcTask Inputs/GVL_iXlinker.EtherCAT_Master_EMxxxx.Beckhoff_EM7xxx.A_0002_EM7004_0000_9996.ENC_Inputs_Channel_3.Latch_value <-> ENC Inputs Channel 3/Latch value
//     PlcTask Inputs/GVL_iXlinker.EtherCAT_Master_EMxxxx.Beckhoff_EM7xxx.A_0002_EM7004_0000_9996.ENC_Inputs_Channel_4.Latch_value <-> ENC Inputs Channel 4/Latch value
//     PlcTask Inputs/GVL_iXlinker.EtherCAT_Master_EMxxxx.Beckhoff_EM7xxx.A_0002_EM7004_0000_9996.PLS_Inputs.PLS_Enabled <-> PLS Inputs/PLS Enabled
//     PlcTask Inputs/GVL_iXlinker.EtherCAT_Master_EMxxxx.Beckhoff_EM7xxx.A_0002_EM7004_0000_9996.PLS_Inputs.Unequal_SI_0 <-> PLS Inputs/Unequal SI:0
//     PlcTask Outputs/GVL_iXlinker.EtherCAT_Master_EMxxxx.Beckhoff_EM7xxx.A_0002_EM7004_0000_9996.DO_Outputs.Output[0] <-> DO Outputs/Output 0
//     PlcTask Outputs/GVL_iXlinker.EtherCAT_Master_EMxxxx.Beckhoff_EM7xxx.A_0002_EM7004_0000_9996.DO_Outputs.Output[1] <-> DO Outputs/Output 1
//     PlcTask Outputs/GVL_iXlinker.EtherCAT_Master_EMxxxx.Beckhoff_EM7xxx.A_0002_EM7004_0000_9996.DO_Outputs.Output[2] <-> DO Outputs/Output 2
//     PlcTask Outputs/GVL_iXlinker.EtherCAT_Master_EMxxxx.Beckhoff_EM7xxx.A_0002_EM7004_0000_9996.DO_Outputs.Output[3] <-> DO Outputs/Output 3
//     PlcTask Outputs/GVL_iXlinker.EtherCAT_Master_EMxxxx.Beckhoff_EM7xxx.A_0002_EM7004_0000_9996.DO_Outputs.Output[4] <-> DO Outputs/Output 4
//     PlcTask Outputs/GVL_iXlinker.EtherCAT_Master_EMxxxx.Beckhoff_EM7xxx.A_0002_EM7004_0000_9996.DO_Outputs.Output[5] <-> DO Outputs/Output 5
//     PlcTask Outputs/GVL_iXlinker.EtherCAT_Master_EMxxxx.Beckhoff_EM7xxx.A_0002_EM7004_0000_9996.DO_Outputs.Output[6] <-> DO Outputs/Output 6
//     PlcTask Outputs/GVL_iXlinker.EtherCAT_Master_EMxxxx.Beckhoff_EM7xxx.A_0002_EM7004_0000_9996.DO_Outputs.Output[7] <-> DO Outputs/Output 7
//     PlcTask Outputs/GVL_iXlinker.EtherCAT_Master_EMxxxx.Beckhoff_EM7xxx.A_0002_EM7004_0000_9996.DO_Outputs.Output[8] <-> DO Outputs/Output 8
//     PlcTask Outputs/GVL_iXlinker.EtherCAT_Master_EMxxxx.Beckhoff_EM7xxx.A_0002_EM7004_0000_9996.DO_Outputs.Output[9] <-> DO Outputs/Output 9
//     PlcTask Outputs/GVL_iXlinker.EtherCAT_Master_EMxxxx.Beckhoff_EM7xxx.A_0002_EM7004_0000_9996.DO_Outputs.Output[10] <-> DO Outputs/Output 10
//     PlcTask Outputs/GVL_iXlinker.EtherCAT_Master_EMxxxx.Beckhoff_EM7xxx.A_0002_EM7004_0000_9996.DO_Outputs.Output[11] <-> DO Outputs/Output 11
//     PlcTask Outputs/GVL_iXlinker.EtherCAT_Master_EMxxxx.Beckhoff_EM7xxx.A_0002_EM7004_0000_9996.DO_Outputs.Output[12] <-> DO Outputs/Output 12
//     PlcTask Outputs/GVL_iXlinker.EtherCAT_Master_EMxxxx.Beckhoff_EM7xxx.A_0002_EM7004_0000_9996.DO_Outputs.Output[13] <-> DO Outputs/Output 13
//     PlcTask Outputs/GVL_iXlinker.EtherCAT_Master_EMxxxx.Beckhoff_EM7xxx.A_0002_EM7004_0000_9996.DO_Outputs.Output[14] <-> DO Outputs/Output 14
//     PlcTask Outputs/GVL_iXlinker.EtherCAT_Master_EMxxxx.Beckhoff_EM7xxx.A_0002_EM7004_0000_9996.DO_Outputs.Output[15] <-> DO Outputs/Output 15
//     PlcTask Outputs/GVL_iXlinker.EtherCAT_Master_EMxxxx.Beckhoff_EM7xxx.A_0002_EM7004_0000_9996.AO_Outputs_Channel_1.Analog_output <-> AO Outputs Channel 1/Analog output
//     PlcTask Outputs/GVL_iXlinker.EtherCAT_Master_EMxxxx.Beckhoff_EM7xxx.A_0002_EM7004_0000_9996.AO_Outputs_Channel_2.Analog_output <-> AO Outputs Channel 2/Analog output
//     PlcTask Outputs/GVL_iXlinker.EtherCAT_Master_EMxxxx.Beckhoff_EM7xxx.A_0002_EM7004_0000_9996.AO_Outputs_Channel_3.Analog_output <-> AO Outputs Channel 3/Analog output
//     PlcTask Outputs/GVL_iXlinker.EtherCAT_Master_EMxxxx.Beckhoff_EM7xxx.A_0002_EM7004_0000_9996.AO_Outputs_Channel_4.Analog_output <-> AO Outputs Channel 4/Analog output
//     PlcTask Outputs/GVL_iXlinker.EtherCAT_Master_EMxxxx.Beckhoff_EM7xxx.A_0002_EM7004_0000_9996.ENC_Outputs_Channel_1.Enable_latch_extern_on_positive_edge <-> ENC Outputs Channel 1/Enable latch extern on positive edge
//     PlcTask Outputs/GVL_iXlinker.EtherCAT_Master_EMxxxx.Beckhoff_EM7xxx.A_0002_EM7004_0000_9996.ENC_Outputs_Channel_2.Enable_latch_extern_on_positive_edge <-> ENC Outputs Channel 2/Enable latch extern on positive edge
//     PlcTask Outputs/GVL_iXlinker.EtherCAT_Master_EMxxxx.Beckhoff_EM7xxx.A_0002_EM7004_0000_9996.ENC_Outputs_Channel_3.Enable_latch_extern_on_positive_edge <-> ENC Outputs Channel 3/Enable latch extern on positive edge
//     PlcTask Outputs/GVL_iXlinker.EtherCAT_Master_EMxxxx.Beckhoff_EM7xxx.A_0002_EM7004_0000_9996.ENC_Outputs_Channel_4.Enable_latch_extern_on_positive_edge <-> ENC Outputs Channel 4/Enable latch extern on positive edge
//     PlcTask Outputs/GVL_iXlinker.EtherCAT_Master_EMxxxx.Beckhoff_EM7xxx.A_0002_EM7004_0000_9996.ENC_Outputs_Channel_1.Set_counter <-> ENC Outputs Channel 1/Set counter
//     PlcTask Outputs/GVL_iXlinker.EtherCAT_Master_EMxxxx.Beckhoff_EM7xxx.A_0002_EM7004_0000_9996.ENC_Outputs_Channel_2.Set_counter <-> ENC Outputs Channel 2/Set counter
//     PlcTask Outputs/GVL_iXlinker.EtherCAT_Master_EMxxxx.Beckhoff_EM7xxx.A_0002_EM7004_0000_9996.ENC_Outputs_Channel_3.Set_counter <-> ENC Outputs Channel 3/Set counter
//     PlcTask Outputs/GVL_iXlinker.EtherCAT_Master_EMxxxx.Beckhoff_EM7xxx.A_0002_EM7004_0000_9996.ENC_Outputs_Channel_4.Set_counter <-> ENC Outputs Channel 4/Set counter
//     PlcTask Outputs/GVL_iXlinker.EtherCAT_Master_EMxxxx.Beckhoff_EM7xxx.A_0002_EM7004_0000_9996.ENC_Outputs_Channel_1.Enable_latch_extern_on_negative_edge <-> ENC Outputs Channel 1/Enable latch extern on negative edge
//     PlcTask Outputs/GVL_iXlinker.EtherCAT_Master_EMxxxx.Beckhoff_EM7xxx.A_0002_EM7004_0000_9996.ENC_Outputs_Channel_2.Enable_latch_extern_on_negative_edge <-> ENC Outputs Channel 2/Enable latch extern on negative edge
//     PlcTask Outputs/GVL_iXlinker.EtherCAT_Master_EMxxxx.Beckhoff_EM7xxx.A_0002_EM7004_0000_9996.ENC_Outputs_Channel_3.Enable_latch_extern_on_negative_edge <-> ENC Outputs Channel 3/Enable latch extern on negative edge
//     PlcTask Outputs/GVL_iXlinker.EtherCAT_Master_EMxxxx.Beckhoff_EM7xxx.A_0002_EM7004_0000_9996.ENC_Outputs_Channel_4.Enable_latch_extern_on_negative_edge <-> ENC Outputs Channel 4/Enable latch extern on negative edge
//     PlcTask Outputs/GVL_iXlinker.EtherCAT_Master_EMxxxx.Beckhoff_EM7xxx.A_0002_EM7004_0000_9996.ENC_Outputs_Channel_1.Set_counter_value <-> ENC Outputs Channel 1/Set counter value
//     PlcTask Outputs/GVL_iXlinker.EtherCAT_Master_EMxxxx.Beckhoff_EM7xxx.A_0002_EM7004_0000_9996.ENC_Outputs_Channel_2.Set_counter_value <-> ENC Outputs Channel 2/Set counter value
//     PlcTask Outputs/GVL_iXlinker.EtherCAT_Master_EMxxxx.Beckhoff_EM7xxx.A_0002_EM7004_0000_9996.ENC_Outputs_Channel_3.Set_counter_value <-> ENC Outputs Channel 3/Set counter value
//     PlcTask Outputs/GVL_iXlinker.EtherCAT_Master_EMxxxx.Beckhoff_EM7xxx.A_0002_EM7004_0000_9996.ENC_Outputs_Channel_4.Set_counter_value <-> ENC Outputs Channel 4/Set counter value
//     PlcTask Outputs/GVL_iXlinker.EtherCAT_Master_EMxxxx.Beckhoff_EM7xxx.A_0002_EM7004_0000_9996.PLS_Outputs.Enable_PLS <-> PLS Outputs/Enable PLS
//     PlcTask Inputs/GVL_iXlinker.EtherCAT_Master_EMxxxx.Beckhoff_EM7xxx.A_0002_EM7004_0000_9996.WcState.WcState <-> WcState/WcState
//     PlcTask Inputs/GVL_iXlinker.EtherCAT_Master_EMxxxx.Beckhoff_EM7xxx.A_0002_EM7004_0000_9996.WcState.InputToggle <-> WcState/InputToggle
//     PlcTask Inputs/GVL_iXlinker.EtherCAT_Master_EMxxxx.Beckhoff_EM7xxx.A_0002_EM7004_0000_9996.InfoData.AdsAddr <-> InfoData/AdsAddr
//     PlcTask Inputs/GVL_iXlinker.EtherCAT_Master_EMxxxx.Beckhoff_EM7xxx.A_0002_EM7004_0000_9996.InfoData.State <-> InfoData/State
//   PLC/PLC Instance <-> EtherCAT Master EMxxxx/Beckhoff EM7xxx/A_0003(EM7004-0000-9997)
//     PlcTask Inputs/GVL_iXlinker.EtherCAT_Master_EMxxxx.Beckhoff_EM7xxx.A_0003_EM7004_0000_9997.DI_Inputs.Input[0] <-> DI Inputs/Input 0
//     PlcTask Inputs/GVL_iXlinker.EtherCAT_Master_EMxxxx.Beckhoff_EM7xxx.A_0003_EM7004_0000_9997.DI_Inputs.Input[1] <-> DI Inputs/Input 1
//     PlcTask Inputs/GVL_iXlinker.EtherCAT_Master_EMxxxx.Beckhoff_EM7xxx.A_0003_EM7004_0000_9997.DI_Inputs.Input[2] <-> DI Inputs/Input 2
//     PlcTask Inputs/GVL_iXlinker.EtherCAT_Master_EMxxxx.Beckhoff_EM7xxx.A_0003_EM7004_0000_9997.DI_Inputs.Input[3] <-> DI Inputs/Input 3
//     PlcTask Inputs/GVL_iXlinker.EtherCAT_Master_EMxxxx.Beckhoff_EM7xxx.A_0003_EM7004_0000_9997.DI_Inputs.Input[4] <-> DI Inputs/Input 4
//     PlcTask Inputs/GVL_iXlinker.EtherCAT_Master_EMxxxx.Beckhoff_EM7xxx.A_0003_EM7004_0000_9997.DI_Inputs.Input[5] <-> DI Inputs/Input 5
//     PlcTask Inputs/GVL_iXlinker.EtherCAT_Master_EMxxxx.Beckhoff_EM7xxx.A_0003_EM7004_0000_9997.DI_Inputs.Input[6] <-> DI Inputs/Input 6
//     PlcTask Inputs/GVL_iXlinker.EtherCAT_Master_EMxxxx.Beckhoff_EM7xxx.A_0003_EM7004_0000_9997.DI_Inputs.Input[7] <-> DI Inputs/Input 7
//     PlcTask Inputs/GVL_iXlinker.EtherCAT_Master_EMxxxx.Beckhoff_EM7xxx.A_0003_EM7004_0000_9997.DI_Inputs.Input[8] <-> DI Inputs/Input 8
//     PlcTask Inputs/GVL_iXlinker.EtherCAT_Master_EMxxxx.Beckhoff_EM7xxx.A_0003_EM7004_0000_9997.DI_Inputs.Input[9] <-> DI Inputs/Input 9
//     PlcTask Inputs/GVL_iXlinker.EtherCAT_Master_EMxxxx.Beckhoff_EM7xxx.A_0003_EM7004_0000_9997.DI_Inputs.Input[10] <-> DI Inputs/Input 10
//     PlcTask Inputs/GVL_iXlinker.EtherCAT_Master_EMxxxx.Beckhoff_EM7xxx.A_0003_EM7004_0000_9997.DI_Inputs.Input[11] <-> DI Inputs/Input 11
//     PlcTask Inputs/GVL_iXlinker.EtherCAT_Master_EMxxxx.Beckhoff_EM7xxx.A_0003_EM7004_0000_9997.DI_Inputs.Input[12] <-> DI Inputs/Input 12
//     PlcTask Inputs/GVL_iXlinker.EtherCAT_Master_EMxxxx.Beckhoff_EM7xxx.A_0003_EM7004_0000_9997.DI_Inputs.Input[13] <-> DI Inputs/Input 13
//     PlcTask Inputs/GVL_iXlinker.EtherCAT_Master_EMxxxx.Beckhoff_EM7xxx.A_0003_EM7004_0000_9997.DI_Inputs.Input[14] <-> DI Inputs/Input 14
//     PlcTask Inputs/GVL_iXlinker.EtherCAT_Master_EMxxxx.Beckhoff_EM7xxx.A_0003_EM7004_0000_9997.DI_Inputs.Input[15] <-> DI Inputs/Input 15
//     PlcTask Inputs/GVL_iXlinker.EtherCAT_Master_EMxxxx.Beckhoff_EM7xxx.A_0003_EM7004_0000_9997.ENC_Inputs_Channel_1.Latch_extern_valid <-> ENC Inputs Channel 1/Latch extern valid
//     PlcTask Inputs/GVL_iXlinker.EtherCAT_Master_EMxxxx.Beckhoff_EM7xxx.A_0003_EM7004_0000_9997.ENC_Inputs_Channel_2.Latch_extern_valid <-> ENC Inputs Channel 2/Latch extern valid
//     PlcTask Inputs/GVL_iXlinker.EtherCAT_Master_EMxxxx.Beckhoff_EM7xxx.A_0003_EM7004_0000_9997.ENC_Inputs_Channel_3.Latch_extern_valid <-> ENC Inputs Channel 3/Latch extern valid
//     PlcTask Inputs/GVL_iXlinker.EtherCAT_Master_EMxxxx.Beckhoff_EM7xxx.A_0003_EM7004_0000_9997.ENC_Inputs_Channel_4.Latch_extern_valid <-> ENC Inputs Channel 4/Latch extern valid
//     PlcTask Inputs/GVL_iXlinker.EtherCAT_Master_EMxxxx.Beckhoff_EM7xxx.A_0003_EM7004_0000_9997.ENC_Inputs_Channel_1.Set_counter_done <-> ENC Inputs Channel 1/Set counter done
//     PlcTask Inputs/GVL_iXlinker.EtherCAT_Master_EMxxxx.Beckhoff_EM7xxx.A_0003_EM7004_0000_9997.ENC_Inputs_Channel_2.Set_counter_done <-> ENC Inputs Channel 2/Set counter done
//     PlcTask Inputs/GVL_iXlinker.EtherCAT_Master_EMxxxx.Beckhoff_EM7xxx.A_0003_EM7004_0000_9997.ENC_Inputs_Channel_3.Set_counter_done <-> ENC Inputs Channel 3/Set counter done
//     PlcTask Inputs/GVL_iXlinker.EtherCAT_Master_EMxxxx.Beckhoff_EM7xxx.A_0003_EM7004_0000_9997.ENC_Inputs_Channel_4.Set_counter_done <-> ENC Inputs Channel 4/Set counter done
//     PlcTask Inputs/GVL_iXlinker.EtherCAT_Master_EMxxxx.Beckhoff_EM7xxx.A_0003_EM7004_0000_9997.ENC_Inputs_Channel_1.Status_of_input_A <-> ENC Inputs Channel 1/Status of input A
//     PlcTask Inputs/GVL_iXlinker.EtherCAT_Master_EMxxxx.Beckhoff_EM7xxx.A_0003_EM7004_0000_9997.ENC_Inputs_Channel_2.Status_of_input_A <-> ENC Inputs Channel 2/Status of input A
//     PlcTask Inputs/GVL_iXlinker.EtherCAT_Master_EMxxxx.Beckhoff_EM7xxx.A_0003_EM7004_0000_9997.ENC_Inputs_Channel_3.Status_of_input_A <-> ENC Inputs Channel 3/Status of input A
//     PlcTask Inputs/GVL_iXlinker.EtherCAT_Master_EMxxxx.Beckhoff_EM7xxx.A_0003_EM7004_0000_9997.ENC_Inputs_Channel_4.Status_of_input_A <-> ENC Inputs Channel 4/Status of input A
//     PlcTask Inputs/GVL_iXlinker.EtherCAT_Master_EMxxxx.Beckhoff_EM7xxx.A_0003_EM7004_0000_9997.ENC_Inputs_Channel_1.Status_of_input_B <-> ENC Inputs Channel 1/Status of input B
//     PlcTask Inputs/GVL_iXlinker.EtherCAT_Master_EMxxxx.Beckhoff_EM7xxx.A_0003_EM7004_0000_9997.ENC_Inputs_Channel_2.Status_of_input_B <-> ENC Inputs Channel 2/Status of input B
//     PlcTask Inputs/GVL_iXlinker.EtherCAT_Master_EMxxxx.Beckhoff_EM7xxx.A_0003_EM7004_0000_9997.ENC_Inputs_Channel_3.Status_of_input_B <-> ENC Inputs Channel 3/Status of input B
//     PlcTask Inputs/GVL_iXlinker.EtherCAT_Master_EMxxxx.Beckhoff_EM7xxx.A_0003_EM7004_0000_9997.ENC_Inputs_Channel_4.Status_of_input_B <-> ENC Inputs Channel 4/Status of input B
//     PlcTask Inputs/GVL_iXlinker.EtherCAT_Master_EMxxxx.Beckhoff_EM7xxx.A_0003_EM7004_0000_9997.ENC_Inputs_Channel_1.Status_of_input_gate <-> ENC Inputs Channel 1/Status of input gate
//     PlcTask Inputs/GVL_iXlinker.EtherCAT_Master_EMxxxx.Beckhoff_EM7xxx.A_0003_EM7004_0000_9997.ENC_Inputs_Channel_2.Status_of_input_gate <-> ENC Inputs Channel 2/Status of input gate
//     PlcTask Inputs/GVL_iXlinker.EtherCAT_Master_EMxxxx.Beckhoff_EM7xxx.A_0003_EM7004_0000_9997.ENC_Inputs_Channel_3.Status_of_input_gate <-> ENC Inputs Channel 3/Status of input gate
//     PlcTask Inputs/GVL_iXlinker.EtherCAT_Master_EMxxxx.Beckhoff_EM7xxx.A_0003_EM7004_0000_9997.ENC_Inputs_Channel_4.Status_of_input_gate <-> ENC Inputs Channel 4/Status of input gate
//     PlcTask Inputs/GVL_iXlinker.EtherCAT_Master_EMxxxx.Beckhoff_EM7xxx.A_0003_EM7004_0000_9997.ENC_Inputs_Channel_1.Status_of_extern_latch <-> ENC Inputs Channel 1/Status of extern latch
//     PlcTask Inputs/GVL_iXlinker.EtherCAT_Master_EMxxxx.Beckhoff_EM7xxx.A_0003_EM7004_0000_9997.ENC_Inputs_Channel_2.Status_of_extern_latch <-> ENC Inputs Channel 2/Status of extern latch
//     PlcTask Inputs/GVL_iXlinker.EtherCAT_Master_EMxxxx.Beckhoff_EM7xxx.A_0003_EM7004_0000_9997.ENC_Inputs_Channel_3.Status_of_extern_latch <-> ENC Inputs Channel 3/Status of extern latch
//     PlcTask Inputs/GVL_iXlinker.EtherCAT_Master_EMxxxx.Beckhoff_EM7xxx.A_0003_EM7004_0000_9997.ENC_Inputs_Channel_4.Status_of_extern_latch <-> ENC Inputs Channel 4/Status of extern latch
//     PlcTask Inputs/GVL_iXlinker.EtherCAT_Master_EMxxxx.Beckhoff_EM7xxx.A_0003_EM7004_0000_9997.ENC_Inputs_Channel_1.Counter_value <-> ENC Inputs Channel 1/Counter value
//     PlcTask Inputs/GVL_iXlinker.EtherCAT_Master_EMxxxx.Beckhoff_EM7xxx.A_0003_EM7004_0000_9997.ENC_Inputs_Channel_2.Counter_value <-> ENC Inputs Channel 2/Counter value
//     PlcTask Inputs/GVL_iXlinker.EtherCAT_Master_EMxxxx.Beckhoff_EM7xxx.A_0003_EM7004_0000_9997.ENC_Inputs_Channel_3.Counter_value <-> ENC Inputs Channel 3/Counter value
//     PlcTask Inputs/GVL_iXlinker.EtherCAT_Master_EMxxxx.Beckhoff_EM7xxx.A_0003_EM7004_0000_9997.ENC_Inputs_Channel_4.Counter_value <-> ENC Inputs Channel 4/Counter value
//     PlcTask Inputs/GVL_iXlinker.EtherCAT_Master_EMxxxx.Beckhoff_EM7xxx.A_0003_EM7004_0000_9997.ENC_Inputs_Channel_1.Latch_value <-> ENC Inputs Channel 1/Latch value
//     PlcTask Inputs/GVL_iXlinker.EtherCAT_Master_EMxxxx.Beckhoff_EM7xxx.A_0003_EM7004_0000_9997.ENC_Inputs_Channel_2.Latch_value <-> ENC Inputs Channel 2/Latch value
//     PlcTask Inputs/GVL_iXlinker.EtherCAT_Master_EMxxxx.Beckhoff_EM7xxx.A_0003_EM7004_0000_9997.ENC_Inputs_Channel_3.Latch_value <-> ENC Inputs Channel 3/Latch value
//     PlcTask Inputs/GVL_iXlinker.EtherCAT_Master_EMxxxx.Beckhoff_EM7xxx.A_0003_EM7004_0000_9997.ENC_Inputs_Channel_4.Latch_value <-> ENC Inputs Channel 4/Latch value
//     PlcTask Inputs/GVL_iXlinker.EtherCAT_Master_EMxxxx.Beckhoff_EM7xxx.A_0003_EM7004_0000_9997.PLS_Inputs.PLS_Enabled <-> PLS Inputs/PLS Enabled
//     PlcTask Inputs/GVL_iXlinker.EtherCAT_Master_EMxxxx.Beckhoff_EM7xxx.A_0003_EM7004_0000_9997.PLS_Inputs.Unequal_SI_0 <-> PLS Inputs/Unequal SI:0
//     PlcTask Outputs/GVL_iXlinker.EtherCAT_Master_EMxxxx.Beckhoff_EM7xxx.A_0003_EM7004_0000_9997.DO_Outputs.Output[0] <-> DO Outputs/Output 0
//     PlcTask Outputs/GVL_iXlinker.EtherCAT_Master_EMxxxx.Beckhoff_EM7xxx.A_0003_EM7004_0000_9997.DO_Outputs.Output[1] <-> DO Outputs/Output 1
//     PlcTask Outputs/GVL_iXlinker.EtherCAT_Master_EMxxxx.Beckhoff_EM7xxx.A_0003_EM7004_0000_9997.DO_Outputs.Output[2] <-> DO Outputs/Output 2
//     PlcTask Outputs/GVL_iXlinker.EtherCAT_Master_EMxxxx.Beckhoff_EM7xxx.A_0003_EM7004_0000_9997.DO_Outputs.Output[3] <-> DO Outputs/Output 3
//     PlcTask Outputs/GVL_iXlinker.EtherCAT_Master_EMxxxx.Beckhoff_EM7xxx.A_0003_EM7004_0000_9997.DO_Outputs.Output[4] <-> DO Outputs/Output 4
//     PlcTask Outputs/GVL_iXlinker.EtherCAT_Master_EMxxxx.Beckhoff_EM7xxx.A_0003_EM7004_0000_9997.DO_Outputs.Output[5] <-> DO Outputs/Output 5
//     PlcTask Outputs/GVL_iXlinker.EtherCAT_Master_EMxxxx.Beckhoff_EM7xxx.A_0003_EM7004_0000_9997.DO_Outputs.Output[6] <-> DO Outputs/Output 6
//     PlcTask Outputs/GVL_iXlinker.EtherCAT_Master_EMxxxx.Beckhoff_EM7xxx.A_0003_EM7004_0000_9997.DO_Outputs.Output[7] <-> DO Outputs/Output 7
//     PlcTask Outputs/GVL_iXlinker.EtherCAT_Master_EMxxxx.Beckhoff_EM7xxx.A_0003_EM7004_0000_9997.DO_Outputs.Output[8] <-> DO Outputs/Output 8
//     PlcTask Outputs/GVL_iXlinker.EtherCAT_Master_EMxxxx.Beckhoff_EM7xxx.A_0003_EM7004_0000_9997.DO_Outputs.Output[9] <-> DO Outputs/Output 9
//     PlcTask Outputs/GVL_iXlinker.EtherCAT_Master_EMxxxx.Beckhoff_EM7xxx.A_0003_EM7004_0000_9997.DO_Outputs.Output[10] <-> DO Outputs/Output 10
//     PlcTask Outputs/GVL_iXlinker.EtherCAT_Master_EMxxxx.Beckhoff_EM7xxx.A_0003_EM7004_0000_9997.DO_Outputs.Output[11] <-> DO Outputs/Output 11
//     PlcTask Outputs/GVL_iXlinker.EtherCAT_Master_EMxxxx.Beckhoff_EM7xxx.A_0003_EM7004_0000_9997.DO_Outputs.Output[12] <-> DO Outputs/Output 12
//     PlcTask Outputs/GVL_iXlinker.EtherCAT_Master_EMxxxx.Beckhoff_EM7xxx.A_0003_EM7004_0000_9997.DO_Outputs.Output[13] <-> DO Outputs/Output 13
//     PlcTask Outputs/GVL_iXlinker.EtherCAT_Master_EMxxxx.Beckhoff_EM7xxx.A_0003_EM7004_0000_9997.DO_Outputs.Output[14] <-> DO Outputs/Output 14
//     PlcTask Outputs/GVL_iXlinker.EtherCAT_Master_EMxxxx.Beckhoff_EM7xxx.A_0003_EM7004_0000_9997.DO_Outputs.Output[15] <-> DO Outputs/Output 15
//     PlcTask Outputs/GVL_iXlinker.EtherCAT_Master_EMxxxx.Beckhoff_EM7xxx.A_0003_EM7004_0000_9997.AO_Outputs_Channel_1.Analog_output <-> AO Outputs Channel 1/Analog output
//     PlcTask Outputs/GVL_iXlinker.EtherCAT_Master_EMxxxx.Beckhoff_EM7xxx.A_0003_EM7004_0000_9997.AO_Outputs_Channel_2.Analog_output <-> AO Outputs Channel 2/Analog output
//     PlcTask Outputs/GVL_iXlinker.EtherCAT_Master_EMxxxx.Beckhoff_EM7xxx.A_0003_EM7004_0000_9997.AO_Outputs_Channel_3.Analog_output <-> AO Outputs Channel 3/Analog output
//     PlcTask Outputs/GVL_iXlinker.EtherCAT_Master_EMxxxx.Beckhoff_EM7xxx.A_0003_EM7004_0000_9997.AO_Outputs_Channel_4.Analog_output <-> AO Outputs Channel 4/Analog output
//     PlcTask Outputs/GVL_iXlinker.EtherCAT_Master_EMxxxx.Beckhoff_EM7xxx.A_0003_EM7004_0000_9997.ENC_Outputs_Channel_1.Enable_latch_extern_on_positive_edge <-> ENC Outputs Channel 1/Enable latch extern on positive edge
//     PlcTask Outputs/GVL_iXlinker.EtherCAT_Master_EMxxxx.Beckhoff_EM7xxx.A_0003_EM7004_0000_9997.ENC_Outputs_Channel_2.Enable_latch_extern_on_positive_edge <-> ENC Outputs Channel 2/Enable latch extern on positive edge
//     PlcTask Outputs/GVL_iXlinker.EtherCAT_Master_EMxxxx.Beckhoff_EM7xxx.A_0003_EM7004_0000_9997.ENC_Outputs_Channel_3.Enable_latch_extern_on_positive_edge <-> ENC Outputs Channel 3/Enable latch extern on positive edge
//     PlcTask Outputs/GVL_iXlinker.EtherCAT_Master_EMxxxx.Beckhoff_EM7xxx.A_0003_EM7004_0000_9997.ENC_Outputs_Channel_4.Enable_latch_extern_on_positive_edge <-> ENC Outputs Channel 4/Enable latch extern on positive edge
//     PlcTask Outputs/GVL_iXlinker.EtherCAT_Master_EMxxxx.Beckhoff_EM7xxx.A_0003_EM7004_0000_9997.ENC_Outputs_Channel_1.Set_counter <-> ENC Outputs Channel 1/Set counter
//     PlcTask Outputs/GVL_iXlinker.EtherCAT_Master_EMxxxx.Beckhoff_EM7xxx.A_0003_EM7004_0000_9997.ENC_Outputs_Channel_2.Set_counter <-> ENC Outputs Channel 2/Set counter
//     PlcTask Outputs/GVL_iXlinker.EtherCAT_Master_EMxxxx.Beckhoff_EM7xxx.A_0003_EM7004_0000_9997.ENC_Outputs_Channel_3.Set_counter <-> ENC Outputs Channel 3/Set counter
//     PlcTask Outputs/GVL_iXlinker.EtherCAT_Master_EMxxxx.Beckhoff_EM7xxx.A_0003_EM7004_0000_9997.ENC_Outputs_Channel_4.Set_counter <-> ENC Outputs Channel 4/Set counter
//     PlcTask Outputs/GVL_iXlinker.EtherCAT_Master_EMxxxx.Beckhoff_EM7xxx.A_0003_EM7004_0000_9997.ENC_Outputs_Channel_1.Enable_latch_extern_on_negative_edge <-> ENC Outputs Channel 1/Enable latch extern on negative edge
//     PlcTask Outputs/GVL_iXlinker.EtherCAT_Master_EMxxxx.Beckhoff_EM7xxx.A_0003_EM7004_0000_9997.ENC_Outputs_Channel_2.Enable_latch_extern_on_negative_edge <-> ENC Outputs Channel 2/Enable latch extern on negative edge
//     PlcTask Outputs/GVL_iXlinker.EtherCAT_Master_EMxxxx.Beckhoff_EM7xxx.A_0003_EM7004_0000_9997.ENC_Outputs_Channel_3.Enable_latch_extern_on_negative_edge <-> ENC Outputs Channel 3/Enable latch extern on negative edge
//     PlcTask Outputs/GVL_iXlinker.EtherCAT_Master_EMxxxx.Beckhoff_EM7xxx.A_0003_EM7004_0000_9997.ENC_Outputs_Channel_4.Enable_latch_extern_on_negative_edge <-> ENC Outputs Channel 4/Enable latch extern on negative edge
//     PlcTask Outputs/GVL_iXlinker.EtherCAT_Master_EMxxxx.Beckhoff_EM7xxx.A_0003_EM7004_0000_9997.ENC_Outputs_Channel_1.Set_counter_value <-> ENC Outputs Channel 1/Set counter value
//     PlcTask Outputs/GVL_iXlinker.EtherCAT_Master_EMxxxx.Beckhoff_EM7xxx.A_0003_EM7004_0000_9997.ENC_Outputs_Channel_2.Set_counter_value <-> ENC Outputs Channel 2/Set counter value
//     PlcTask Outputs/GVL_iXlinker.EtherCAT_Master_EMxxxx.Beckhoff_EM7xxx.A_0003_EM7004_0000_9997.ENC_Outputs_Channel_3.Set_counter_value <-> ENC Outputs Channel 3/Set counter value
//     PlcTask Outputs/GVL_iXlinker.EtherCAT_Master_EMxxxx.Beckhoff_EM7xxx.A_0003_EM7004_0000_9997.ENC_Outputs_Channel_4.Set_counter_value <-> ENC Outputs Channel 4/Set counter value
//     PlcTask Outputs/GVL_iXlinker.EtherCAT_Master_EMxxxx.Beckhoff_EM7xxx.A_0003_EM7004_0000_9997.PLS_Outputs.Enable_PLS <-> PLS Outputs/Enable PLS
//     PlcTask Inputs/GVL_iXlinker.EtherCAT_Master_EMxxxx.Beckhoff_EM7xxx.A_0003_EM7004_0000_9997.WcState.WcState <-> WcState/WcState
//     PlcTask Inputs/GVL_iXlinker.EtherCAT_Master_EMxxxx.Beckhoff_EM7xxx.A_0003_EM7004_0000_9997.WcState.InputToggle <-> WcState/InputToggle
//     PlcTask Inputs/GVL_iXlinker.EtherCAT_Master_EMxxxx.Beckhoff_EM7xxx.A_0003_EM7004_0000_9997.InfoData.AdsAddr <-> InfoData/AdsAddr
//     PlcTask Inputs/GVL_iXlinker.EtherCAT_Master_EMxxxx.Beckhoff_EM7xxx.A_0003_EM7004_0000_9997.InfoData.State <-> InfoData/State
//   PLC/PLC Instance <-> EtherCAT Master EMxxxx/Beckhoff EM7xxx/A_0004(EM7004-0000-0016)
//     PlcTask Inputs/GVL_iXlinker.EtherCAT_Master_EMxxxx.Beckhoff_EM7xxx.A_0004_EM7004_0000_0016.DI_Inputs.Input[0] <-> DI Inputs/Input 0
//     PlcTask Inputs/GVL_iXlinker.EtherCAT_Master_EMxxxx.Beckhoff_EM7xxx.A_0004_EM7004_0000_0016.DI_Inputs.Input[1] <-> DI Inputs/Input 1
//     PlcTask Inputs/GVL_iXlinker.EtherCAT_Master_EMxxxx.Beckhoff_EM7xxx.A_0004_EM7004_0000_0016.DI_Inputs.Input[2] <-> DI Inputs/Input 2
//     PlcTask Inputs/GVL_iXlinker.EtherCAT_Master_EMxxxx.Beckhoff_EM7xxx.A_0004_EM7004_0000_0016.DI_Inputs.Input[3] <-> DI Inputs/Input 3
//     PlcTask Inputs/GVL_iXlinker.EtherCAT_Master_EMxxxx.Beckhoff_EM7xxx.A_0004_EM7004_0000_0016.DI_Inputs.Input[4] <-> DI Inputs/Input 4
//     PlcTask Inputs/GVL_iXlinker.EtherCAT_Master_EMxxxx.Beckhoff_EM7xxx.A_0004_EM7004_0000_0016.DI_Inputs.Input[5] <-> DI Inputs/Input 5
//     PlcTask Inputs/GVL_iXlinker.EtherCAT_Master_EMxxxx.Beckhoff_EM7xxx.A_0004_EM7004_0000_0016.DI_Inputs.Input[6] <-> DI Inputs/Input 6
//     PlcTask Inputs/GVL_iXlinker.EtherCAT_Master_EMxxxx.Beckhoff_EM7xxx.A_0004_EM7004_0000_0016.DI_Inputs.Input[7] <-> DI Inputs/Input 7
//     PlcTask Inputs/GVL_iXlinker.EtherCAT_Master_EMxxxx.Beckhoff_EM7xxx.A_0004_EM7004_0000_0016.DI_Inputs.Input[8] <-> DI Inputs/Input 8
//     PlcTask Inputs/GVL_iXlinker.EtherCAT_Master_EMxxxx.Beckhoff_EM7xxx.A_0004_EM7004_0000_0016.DI_Inputs.Input[9] <-> DI Inputs/Input 9
//     PlcTask Inputs/GVL_iXlinker.EtherCAT_Master_EMxxxx.Beckhoff_EM7xxx.A_0004_EM7004_0000_0016.DI_Inputs.Input[10] <-> DI Inputs/Input 10
//     PlcTask Inputs/GVL_iXlinker.EtherCAT_Master_EMxxxx.Beckhoff_EM7xxx.A_0004_EM7004_0000_0016.DI_Inputs.Input[11] <-> DI Inputs/Input 11
//     PlcTask Inputs/GVL_iXlinker.EtherCAT_Master_EMxxxx.Beckhoff_EM7xxx.A_0004_EM7004_0000_0016.DI_Inputs.Input[12] <-> DI Inputs/Input 12
//     PlcTask Inputs/GVL_iXlinker.EtherCAT_Master_EMxxxx.Beckhoff_EM7xxx.A_0004_EM7004_0000_0016.DI_Inputs.Input[13] <-> DI Inputs/Input 13
//     PlcTask Inputs/GVL_iXlinker.EtherCAT_Master_EMxxxx.Beckhoff_EM7xxx.A_0004_EM7004_0000_0016.DI_Inputs.Input[14] <-> DI Inputs/Input 14
//     PlcTask Inputs/GVL_iXlinker.EtherCAT_Master_EMxxxx.Beckhoff_EM7xxx.A_0004_EM7004_0000_0016.DI_Inputs.Input[15] <-> DI Inputs/Input 15
//     PlcTask Inputs/GVL_iXlinker.EtherCAT_Master_EMxxxx.Beckhoff_EM7xxx.A_0004_EM7004_0000_0016.ENC_Inputs_Channel_1.Latch_extern_valid <-> ENC Inputs Channel 1/Latch extern valid
//     PlcTask Inputs/GVL_iXlinker.EtherCAT_Master_EMxxxx.Beckhoff_EM7xxx.A_0004_EM7004_0000_0016.ENC_Inputs_Channel_2.Latch_extern_valid <-> ENC Inputs Channel 2/Latch extern valid
//     PlcTask Inputs/GVL_iXlinker.EtherCAT_Master_EMxxxx.Beckhoff_EM7xxx.A_0004_EM7004_0000_0016.ENC_Inputs_Channel_3.Latch_extern_valid <-> ENC Inputs Channel 3/Latch extern valid
//     PlcTask Inputs/GVL_iXlinker.EtherCAT_Master_EMxxxx.Beckhoff_EM7xxx.A_0004_EM7004_0000_0016.ENC_Inputs_Channel_4.Latch_extern_valid <-> ENC Inputs Channel 4/Latch extern valid
//     PlcTask Inputs/GVL_iXlinker.EtherCAT_Master_EMxxxx.Beckhoff_EM7xxx.A_0004_EM7004_0000_0016.ENC_Inputs_Channel_1.Set_counter_done <-> ENC Inputs Channel 1/Set counter done
//     PlcTask Inputs/GVL_iXlinker.EtherCAT_Master_EMxxxx.Beckhoff_EM7xxx.A_0004_EM7004_0000_0016.ENC_Inputs_Channel_2.Set_counter_done <-> ENC Inputs Channel 2/Set counter done
//     PlcTask Inputs/GVL_iXlinker.EtherCAT_Master_EMxxxx.Beckhoff_EM7xxx.A_0004_EM7004_0000_0016.ENC_Inputs_Channel_3.Set_counter_done <-> ENC Inputs Channel 3/Set counter done
//     PlcTask Inputs/GVL_iXlinker.EtherCAT_Master_EMxxxx.Beckhoff_EM7xxx.A_0004_EM7004_0000_0016.ENC_Inputs_Channel_4.Set_counter_done <-> ENC Inputs Channel 4/Set counter done
//     PlcTask Inputs/GVL_iXlinker.EtherCAT_Master_EMxxxx.Beckhoff_EM7xxx.A_0004_EM7004_0000_0016.ENC_Inputs_Channel_1.Status_of_input_A <-> ENC Inputs Channel 1/Status of input A
//     PlcTask Inputs/GVL_iXlinker.EtherCAT_Master_EMxxxx.Beckhoff_EM7xxx.A_0004_EM7004_0000_0016.ENC_Inputs_Channel_2.Status_of_input_A <-> ENC Inputs Channel 2/Status of input A
//     PlcTask Inputs/GVL_iXlinker.EtherCAT_Master_EMxxxx.Beckhoff_EM7xxx.A_0004_EM7004_0000_0016.ENC_Inputs_Channel_3.Status_of_input_A <-> ENC Inputs Channel 3/Status of input A
//     PlcTask Inputs/GVL_iXlinker.EtherCAT_Master_EMxxxx.Beckhoff_EM7xxx.A_0004_EM7004_0000_0016.ENC_Inputs_Channel_4.Status_of_input_A <-> ENC Inputs Channel 4/Status of input A
//     PlcTask Inputs/GVL_iXlinker.EtherCAT_Master_EMxxxx.Beckhoff_EM7xxx.A_0004_EM7004_0000_0016.ENC_Inputs_Channel_1.Status_of_input_B <-> ENC Inputs Channel 1/Status of input B
//     PlcTask Inputs/GVL_iXlinker.EtherCAT_Master_EMxxxx.Beckhoff_EM7xxx.A_0004_EM7004_0000_0016.ENC_Inputs_Channel_2.Status_of_input_B <-> ENC Inputs Channel 2/Status of input B
//     PlcTask Inputs/GVL_iXlinker.EtherCAT_Master_EMxxxx.Beckhoff_EM7xxx.A_0004_EM7004_0000_0016.ENC_Inputs_Channel_3.Status_of_input_B <-> ENC Inputs Channel 3/Status of input B
//     PlcTask Inputs/GVL_iXlinker.EtherCAT_Master_EMxxxx.Beckhoff_EM7xxx.A_0004_EM7004_0000_0016.ENC_Inputs_Channel_4.Status_of_input_B <-> ENC Inputs Channel 4/Status of input B
//     PlcTask Inputs/GVL_iXlinker.EtherCAT_Master_EMxxxx.Beckhoff_EM7xxx.A_0004_EM7004_0000_0016.ENC_Inputs_Channel_1.Status_of_input_gate <-> ENC Inputs Channel 1/Status of input gate
//     PlcTask Inputs/GVL_iXlinker.EtherCAT_Master_EMxxxx.Beckhoff_EM7xxx.A_0004_EM7004_0000_0016.ENC_Inputs_Channel_2.Status_of_input_gate <-> ENC Inputs Channel 2/Status of input gate
//     PlcTask Inputs/GVL_iXlinker.EtherCAT_Master_EMxxxx.Beckhoff_EM7xxx.A_0004_EM7004_0000_0016.ENC_Inputs_Channel_3.Status_of_input_gate <-> ENC Inputs Channel 3/Status of input gate
//     PlcTask Inputs/GVL_iXlinker.EtherCAT_Master_EMxxxx.Beckhoff_EM7xxx.A_0004_EM7004_0000_0016.ENC_Inputs_Channel_4.Status_of_input_gate <-> ENC Inputs Channel 4/Status of input gate
//     PlcTask Inputs/GVL_iXlinker.EtherCAT_Master_EMxxxx.Beckhoff_EM7xxx.A_0004_EM7004_0000_0016.ENC_Inputs_Channel_1.Status_of_extern_latch <-> ENC Inputs Channel 1/Status of extern latch
//     PlcTask Inputs/GVL_iXlinker.EtherCAT_Master_EMxxxx.Beckhoff_EM7xxx.A_0004_EM7004_0000_0016.ENC_Inputs_Channel_2.Status_of_extern_latch <-> ENC Inputs Channel 2/Status of extern latch
//     PlcTask Inputs/GVL_iXlinker.EtherCAT_Master_EMxxxx.Beckhoff_EM7xxx.A_0004_EM7004_0000_0016.ENC_Inputs_Channel_3.Status_of_extern_latch <-> ENC Inputs Channel 3/Status of extern latch
//     PlcTask Inputs/GVL_iXlinker.EtherCAT_Master_EMxxxx.Beckhoff_EM7xxx.A_0004_EM7004_0000_0016.ENC_Inputs_Channel_4.Status_of_extern_latch <-> ENC Inputs Channel 4/Status of extern latch
//     PlcTask Inputs/GVL_iXlinker.EtherCAT_Master_EMxxxx.Beckhoff_EM7xxx.A_0004_EM7004_0000_0016.ENC_Inputs_Channel_1.TxPDO_Toggle <-> ENC Inputs Channel 1/TxPDO Toggle
//     PlcTask Inputs/GVL_iXlinker.EtherCAT_Master_EMxxxx.Beckhoff_EM7xxx.A_0004_EM7004_0000_0016.ENC_Inputs_Channel_2.TxPDO_Toggle <-> ENC Inputs Channel 2/TxPDO Toggle
//     PlcTask Inputs/GVL_iXlinker.EtherCAT_Master_EMxxxx.Beckhoff_EM7xxx.A_0004_EM7004_0000_0016.ENC_Inputs_Channel_3.TxPDO_Toggle <-> ENC Inputs Channel 3/TxPDO Toggle
//     PlcTask Inputs/GVL_iXlinker.EtherCAT_Master_EMxxxx.Beckhoff_EM7xxx.A_0004_EM7004_0000_0016.ENC_Inputs_Channel_4.TxPDO_Toggle <-> ENC Inputs Channel 4/TxPDO Toggle
//     PlcTask Inputs/GVL_iXlinker.EtherCAT_Master_EMxxxx.Beckhoff_EM7xxx.A_0004_EM7004_0000_0016.ENC_Inputs_Channel_1.Counter_value <-> ENC Inputs Channel 1/Counter value
//     PlcTask Inputs/GVL_iXlinker.EtherCAT_Master_EMxxxx.Beckhoff_EM7xxx.A_0004_EM7004_0000_0016.ENC_Inputs_Channel_2.Counter_value <-> ENC Inputs Channel 2/Counter value
//     PlcTask Inputs/GVL_iXlinker.EtherCAT_Master_EMxxxx.Beckhoff_EM7xxx.A_0004_EM7004_0000_0016.ENC_Inputs_Channel_3.Counter_value <-> ENC Inputs Channel 3/Counter value
//     PlcTask Inputs/GVL_iXlinker.EtherCAT_Master_EMxxxx.Beckhoff_EM7xxx.A_0004_EM7004_0000_0016.ENC_Inputs_Channel_4.Counter_value <-> ENC Inputs Channel 4/Counter value
//     PlcTask Inputs/GVL_iXlinker.EtherCAT_Master_EMxxxx.Beckhoff_EM7xxx.A_0004_EM7004_0000_0016.ENC_Inputs_Channel_1.Latch_value <-> ENC Inputs Channel 1/Latch value
//     PlcTask Inputs/GVL_iXlinker.EtherCAT_Master_EMxxxx.Beckhoff_EM7xxx.A_0004_EM7004_0000_0016.ENC_Inputs_Channel_2.Latch_value <-> ENC Inputs Channel 2/Latch value
//     PlcTask Inputs/GVL_iXlinker.EtherCAT_Master_EMxxxx.Beckhoff_EM7xxx.A_0004_EM7004_0000_0016.ENC_Inputs_Channel_3.Latch_value <-> ENC Inputs Channel 3/Latch value
//     PlcTask Inputs/GVL_iXlinker.EtherCAT_Master_EMxxxx.Beckhoff_EM7xxx.A_0004_EM7004_0000_0016.ENC_Inputs_Channel_4.Latch_value <-> ENC Inputs Channel 4/Latch value
//     PlcTask Inputs/GVL_iXlinker.EtherCAT_Master_EMxxxx.Beckhoff_EM7xxx.A_0004_EM7004_0000_0016.PLS_Inputs.PLS_Enabled <-> PLS Inputs/PLS Enabled
//     PlcTask Inputs/GVL_iXlinker.EtherCAT_Master_EMxxxx.Beckhoff_EM7xxx.A_0004_EM7004_0000_0016.PLS_Inputs.Unequal_SI_0 <-> PLS Inputs/Unequal SI:0
//     PlcTask Outputs/GVL_iXlinker.EtherCAT_Master_EMxxxx.Beckhoff_EM7xxx.A_0004_EM7004_0000_0016.DO_Outputs.Output[0] <-> DO Outputs/Output 0
//     PlcTask Outputs/GVL_iXlinker.EtherCAT_Master_EMxxxx.Beckhoff_EM7xxx.A_0004_EM7004_0000_0016.DO_Outputs.Output[1] <-> DO Outputs/Output 1
//     PlcTask Outputs/GVL_iXlinker.EtherCAT_Master_EMxxxx.Beckhoff_EM7xxx.A_0004_EM7004_0000_0016.DO_Outputs.Output[2] <-> DO Outputs/Output 2
//     PlcTask Outputs/GVL_iXlinker.EtherCAT_Master_EMxxxx.Beckhoff_EM7xxx.A_0004_EM7004_0000_0016.DO_Outputs.Output[3] <-> DO Outputs/Output 3
//     PlcTask Outputs/GVL_iXlinker.EtherCAT_Master_EMxxxx.Beckhoff_EM7xxx.A_0004_EM7004_0000_0016.DO_Outputs.Output[4] <-> DO Outputs/Output 4
//     PlcTask Outputs/GVL_iXlinker.EtherCAT_Master_EMxxxx.Beckhoff_EM7xxx.A_0004_EM7004_0000_0016.DO_Outputs.Output[5] <-> DO Outputs/Output 5
//     PlcTask Outputs/GVL_iXlinker.EtherCAT_Master_EMxxxx.Beckhoff_EM7xxx.A_0004_EM7004_0000_0016.DO_Outputs.Output[6] <-> DO Outputs/Output 6
//     PlcTask Outputs/GVL_iXlinker.EtherCAT_Master_EMxxxx.Beckhoff_EM7xxx.A_0004_EM7004_0000_0016.DO_Outputs.Output[7] <-> DO Outputs/Output 7
//     PlcTask Outputs/GVL_iXlinker.EtherCAT_Master_EMxxxx.Beckhoff_EM7xxx.A_0004_EM7004_0000_0016.DO_Outputs.Output[8] <-> DO Outputs/Output 8
//     PlcTask Outputs/GVL_iXlinker.EtherCAT_Master_EMxxxx.Beckhoff_EM7xxx.A_0004_EM7004_0000_0016.DO_Outputs.Output[9] <-> DO Outputs/Output 9
//     PlcTask Outputs/GVL_iXlinker.EtherCAT_Master_EMxxxx.Beckhoff_EM7xxx.A_0004_EM7004_0000_0016.DO_Outputs.Output[10] <-> DO Outputs/Output 10
//     PlcTask Outputs/GVL_iXlinker.EtherCAT_Master_EMxxxx.Beckhoff_EM7xxx.A_0004_EM7004_0000_0016.DO_Outputs.Output[11] <-> DO Outputs/Output 11
//     PlcTask Outputs/GVL_iXlinker.EtherCAT_Master_EMxxxx.Beckhoff_EM7xxx.A_0004_EM7004_0000_0016.DO_Outputs.Output[12] <-> DO Outputs/Output 12
//     PlcTask Outputs/GVL_iXlinker.EtherCAT_Master_EMxxxx.Beckhoff_EM7xxx.A_0004_EM7004_0000_0016.DO_Outputs.Output[13] <-> DO Outputs/Output 13
//     PlcTask Outputs/GVL_iXlinker.EtherCAT_Master_EMxxxx.Beckhoff_EM7xxx.A_0004_EM7004_0000_0016.DO_Outputs.Output[14] <-> DO Outputs/Output 14
//     PlcTask Outputs/GVL_iXlinker.EtherCAT_Master_EMxxxx.Beckhoff_EM7xxx.A_0004_EM7004_0000_0016.DO_Outputs.Output[15] <-> DO Outputs/Output 15
//     PlcTask Outputs/GVL_iXlinker.EtherCAT_Master_EMxxxx.Beckhoff_EM7xxx.A_0004_EM7004_0000_0016.AO_Outputs_Channel_1.Analog_output <-> AO Outputs Channel 1/Analog output
//     PlcTask Outputs/GVL_iXlinker.EtherCAT_Master_EMxxxx.Beckhoff_EM7xxx.A_0004_EM7004_0000_0016.AO_Outputs_Channel_2.Analog_output <-> AO Outputs Channel 2/Analog output
//     PlcTask Outputs/GVL_iXlinker.EtherCAT_Master_EMxxxx.Beckhoff_EM7xxx.A_0004_EM7004_0000_0016.AO_Outputs_Channel_3.Analog_output <-> AO Outputs Channel 3/Analog output
//     PlcTask Outputs/GVL_iXlinker.EtherCAT_Master_EMxxxx.Beckhoff_EM7xxx.A_0004_EM7004_0000_0016.AO_Outputs_Channel_4.Analog_output <-> AO Outputs Channel 4/Analog output
//     PlcTask Outputs/GVL_iXlinker.EtherCAT_Master_EMxxxx.Beckhoff_EM7xxx.A_0004_EM7004_0000_0016.ENC_Outputs_Channel_1.Enable_latch_extern_on_positive_edge <-> ENC Outputs Channel 1/Enable latch extern on positive edge
//     PlcTask Outputs/GVL_iXlinker.EtherCAT_Master_EMxxxx.Beckhoff_EM7xxx.A_0004_EM7004_0000_0016.ENC_Outputs_Channel_2.Enable_latch_extern_on_positive_edge <-> ENC Outputs Channel 2/Enable latch extern on positive edge
//     PlcTask Outputs/GVL_iXlinker.EtherCAT_Master_EMxxxx.Beckhoff_EM7xxx.A_0004_EM7004_0000_0016.ENC_Outputs_Channel_3.Enable_latch_extern_on_positive_edge <-> ENC Outputs Channel 3/Enable latch extern on positive edge
//     PlcTask Outputs/GVL_iXlinker.EtherCAT_Master_EMxxxx.Beckhoff_EM7xxx.A_0004_EM7004_0000_0016.ENC_Outputs_Channel_4.Enable_latch_extern_on_positive_edge <-> ENC Outputs Channel 4/Enable latch extern on positive edge
//     PlcTask Outputs/GVL_iXlinker.EtherCAT_Master_EMxxxx.Beckhoff_EM7xxx.A_0004_EM7004_0000_0016.ENC_Outputs_Channel_1.Set_counter <-> ENC Outputs Channel 1/Set counter
//     PlcTask Outputs/GVL_iXlinker.EtherCAT_Master_EMxxxx.Beckhoff_EM7xxx.A_0004_EM7004_0000_0016.ENC_Outputs_Channel_2.Set_counter <-> ENC Outputs Channel 2/Set counter
//     PlcTask Outputs/GVL_iXlinker.EtherCAT_Master_EMxxxx.Beckhoff_EM7xxx.A_0004_EM7004_0000_0016.ENC_Outputs_Channel_3.Set_counter <-> ENC Outputs Channel 3/Set counter
//     PlcTask Outputs/GVL_iXlinker.EtherCAT_Master_EMxxxx.Beckhoff_EM7xxx.A_0004_EM7004_0000_0016.ENC_Outputs_Channel_4.Set_counter <-> ENC Outputs Channel 4/Set counter
//     PlcTask Outputs/GVL_iXlinker.EtherCAT_Master_EMxxxx.Beckhoff_EM7xxx.A_0004_EM7004_0000_0016.ENC_Outputs_Channel_1.Enable_latch_extern_on_negative_edge <-> ENC Outputs Channel 1/Enable latch extern on negative edge
//     PlcTask Outputs/GVL_iXlinker.EtherCAT_Master_EMxxxx.Beckhoff_EM7xxx.A_0004_EM7004_0000_0016.ENC_Outputs_Channel_2.Enable_latch_extern_on_negative_edge <-> ENC Outputs Channel 2/Enable latch extern on negative edge
//     PlcTask Outputs/GVL_iXlinker.EtherCAT_Master_EMxxxx.Beckhoff_EM7xxx.A_0004_EM7004_0000_0016.ENC_Outputs_Channel_3.Enable_latch_extern_on_negative_edge <-> ENC Outputs Channel 3/Enable latch extern on negative edge
//     PlcTask Outputs/GVL_iXlinker.EtherCAT_Master_EMxxxx.Beckhoff_EM7xxx.A_0004_EM7004_0000_0016.ENC_Outputs_Channel_4.Enable_latch_extern_on_negative_edge <-> ENC Outputs Channel 4/Enable latch extern on negative edge
//     PlcTask Outputs/GVL_iXlinker.EtherCAT_Master_EMxxxx.Beckhoff_EM7xxx.A_0004_EM7004_0000_0016.ENC_Outputs_Channel_1.Set_counter_value <-> ENC Outputs Channel 1/Set counter value
//     PlcTask Outputs/GVL_iXlinker.EtherCAT_Master_EMxxxx.Beckhoff_EM7xxx.A_0004_EM7004_0000_0016.ENC_Outputs_Channel_2.Set_counter_value <-> ENC Outputs Channel 2/Set counter value
//     PlcTask Outputs/GVL_iXlinker.EtherCAT_Master_EMxxxx.Beckhoff_EM7xxx.A_0004_EM7004_0000_0016.ENC_Outputs_Channel_3.Set_counter_value <-> ENC Outputs Channel 3/Set counter value
//     PlcTask Outputs/GVL_iXlinker.EtherCAT_Master_EMxxxx.Beckhoff_EM7xxx.A_0004_EM7004_0000_0016.ENC_Outputs_Channel_4.Set_counter_value <-> ENC Outputs Channel 4/Set counter value
//     PlcTask Outputs/GVL_iXlinker.EtherCAT_Master_EMxxxx.Beckhoff_EM7xxx.A_0004_EM7004_0000_0016.PLS_Outputs.Enable_PLS <-> PLS Outputs/Enable PLS
//     PlcTask Inputs/GVL_iXlinker.EtherCAT_Master_EMxxxx.Beckhoff_EM7xxx.A_0004_EM7004_0000_0016.WcState.WcState <-> WcState/WcState
//     PlcTask Inputs/GVL_iXlinker.EtherCAT_Master_EMxxxx.Beckhoff_EM7xxx.A_0004_EM7004_0000_0016.WcState.InputToggle <-> WcState/InputToggle
//     PlcTask Inputs/GVL_iXlinker.EtherCAT_Master_EMxxxx.Beckhoff_EM7xxx.A_0004_EM7004_0000_0016.InfoData.AdsAddr <-> InfoData/AdsAddr
//     PlcTask Inputs/GVL_iXlinker.EtherCAT_Master_EMxxxx.Beckhoff_EM7xxx.A_0004_EM7004_0000_0016.InfoData.State <-> InfoData/State
//   PLC/PLC Instance <-> EtherCAT Master EMxxxx/Beckhoff EM7xxx/A_0005(EM7004-0000-0017)
//     PlcTask Inputs/GVL_iXlinker.EtherCAT_Master_EMxxxx.Beckhoff_EM7xxx.A_0005_EM7004_0000_0017.DI_Inputs.Input/Input_0 <-> DI Inputs/Input/Input 0
//     PlcTask Inputs/GVL_iXlinker.EtherCAT_Master_EMxxxx.Beckhoff_EM7xxx.A_0005_EM7004_0000_0017.DI_Inputs.Input/Input_1 <-> DI Inputs/Input/Input 1
//     PlcTask Inputs/GVL_iXlinker.EtherCAT_Master_EMxxxx.Beckhoff_EM7xxx.A_0005_EM7004_0000_0017.DI_Inputs.Input/Input_2 <-> DI Inputs/Input/Input 2
//     PlcTask Inputs/GVL_iXlinker.EtherCAT_Master_EMxxxx.Beckhoff_EM7xxx.A_0005_EM7004_0000_0017.DI_Inputs.Input/Input_3 <-> DI Inputs/Input/Input 3
//     PlcTask Inputs/GVL_iXlinker.EtherCAT_Master_EMxxxx.Beckhoff_EM7xxx.A_0005_EM7004_0000_0017.DI_Inputs.Input/Input_4 <-> DI Inputs/Input/Input 4
//     PlcTask Inputs/GVL_iXlinker.EtherCAT_Master_EMxxxx.Beckhoff_EM7xxx.A_0005_EM7004_0000_0017.DI_Inputs.Input/Input_5 <-> DI Inputs/Input/Input 5
//     PlcTask Inputs/GVL_iXlinker.EtherCAT_Master_EMxxxx.Beckhoff_EM7xxx.A_0005_EM7004_0000_0017.DI_Inputs.Input/Input_6 <-> DI Inputs/Input/Input 6
//     PlcTask Inputs/GVL_iXlinker.EtherCAT_Master_EMxxxx.Beckhoff_EM7xxx.A_0005_EM7004_0000_0017.DI_Inputs.Input/Input_7 <-> DI Inputs/Input/Input 7
//     PlcTask Inputs/GVL_iXlinker.EtherCAT_Master_EMxxxx.Beckhoff_EM7xxx.A_0005_EM7004_0000_0017.DI_Inputs.Input/Input_8 <-> DI Inputs/Input/Input 8
//     PlcTask Inputs/GVL_iXlinker.EtherCAT_Master_EMxxxx.Beckhoff_EM7xxx.A_0005_EM7004_0000_0017.DI_Inputs.Input/Input_9 <-> DI Inputs/Input/Input 9
//     PlcTask Inputs/GVL_iXlinker.EtherCAT_Master_EMxxxx.Beckhoff_EM7xxx.A_0005_EM7004_0000_0017.DI_Inputs.Input/Input_10 <-> DI Inputs/Input/Input 10
//     PlcTask Inputs/GVL_iXlinker.EtherCAT_Master_EMxxxx.Beckhoff_EM7xxx.A_0005_EM7004_0000_0017.DI_Inputs.Input/Input_11 <-> DI Inputs/Input/Input 11
//     PlcTask Inputs/GVL_iXlinker.EtherCAT_Master_EMxxxx.Beckhoff_EM7xxx.A_0005_EM7004_0000_0017.DI_Inputs.Input/Input_12 <-> DI Inputs/Input/Input 12
//     PlcTask Inputs/GVL_iXlinker.EtherCAT_Master_EMxxxx.Beckhoff_EM7xxx.A_0005_EM7004_0000_0017.DI_Inputs.Input/Input_13 <-> DI Inputs/Input/Input 13
//     PlcTask Inputs/GVL_iXlinker.EtherCAT_Master_EMxxxx.Beckhoff_EM7xxx.A_0005_EM7004_0000_0017.DI_Inputs.Input/Input_14 <-> DI Inputs/Input/Input 14
//     PlcTask Inputs/GVL_iXlinker.EtherCAT_Master_EMxxxx.Beckhoff_EM7xxx.A_0005_EM7004_0000_0017.DI_Inputs.Input/Input_15 <-> DI Inputs/Input/Input 15
//     PlcTask Inputs/GVL_iXlinker.EtherCAT_Master_EMxxxx.Beckhoff_EM7xxx.A_0005_EM7004_0000_0017.ENC_Inputs_Channel_1.Status/Latch_extern_valid <-> ENC Inputs Channel 1/Status/Latch extern valid
//     PlcTask Inputs/GVL_iXlinker.EtherCAT_Master_EMxxxx.Beckhoff_EM7xxx.A_0005_EM7004_0000_0017.ENC_Inputs_Channel_2.Status/Latch_extern_valid <-> ENC Inputs Channel 2/Status/Latch extern valid
//     PlcTask Inputs/GVL_iXlinker.EtherCAT_Master_EMxxxx.Beckhoff_EM7xxx.A_0005_EM7004_0000_0017.ENC_Inputs_Channel_3.Status/Latch_extern_valid <-> ENC Inputs Channel 3/Status/Latch extern valid
//     PlcTask Inputs/GVL_iXlinker.EtherCAT_Master_EMxxxx.Beckhoff_EM7xxx.A_0005_EM7004_0000_0017.ENC_Inputs_Channel_4.Status/Latch_extern_valid <-> ENC Inputs Channel 4/Status/Latch extern valid
//     PlcTask Inputs/GVL_iXlinker.EtherCAT_Master_EMxxxx.Beckhoff_EM7xxx.A_0005_EM7004_0000_0017.ENC_Inputs_Channel_1.Status/Set_counter_done <-> ENC Inputs Channel 1/Status/Set counter done
//     PlcTask Inputs/GVL_iXlinker.EtherCAT_Master_EMxxxx.Beckhoff_EM7xxx.A_0005_EM7004_0000_0017.ENC_Inputs_Channel_2.Status/Set_counter_done <-> ENC Inputs Channel 2/Status/Set counter done
//     PlcTask Inputs/GVL_iXlinker.EtherCAT_Master_EMxxxx.Beckhoff_EM7xxx.A_0005_EM7004_0000_0017.ENC_Inputs_Channel_3.Status/Set_counter_done <-> ENC Inputs Channel 3/Status/Set counter done
//     PlcTask Inputs/GVL_iXlinker.EtherCAT_Master_EMxxxx.Beckhoff_EM7xxx.A_0005_EM7004_0000_0017.ENC_Inputs_Channel_4.Status/Set_counter_done <-> ENC Inputs Channel 4/Status/Set counter done
//     PlcTask Inputs/GVL_iXlinker.EtherCAT_Master_EMxxxx.Beckhoff_EM7xxx.A_0005_EM7004_0000_0017.ENC_Inputs_Channel_1.Status/Status_of_input_A <-> ENC Inputs Channel 1/Status/Status of input A
//     PlcTask Inputs/GVL_iXlinker.EtherCAT_Master_EMxxxx.Beckhoff_EM7xxx.A_0005_EM7004_0000_0017.ENC_Inputs_Channel_2.Status/Status_of_input_A <-> ENC Inputs Channel 2/Status/Status of input A
//     PlcTask Inputs/GVL_iXlinker.EtherCAT_Master_EMxxxx.Beckhoff_EM7xxx.A_0005_EM7004_0000_0017.ENC_Inputs_Channel_3.Status/Status_of_input_A <-> ENC Inputs Channel 3/Status/Status of input A
//     PlcTask Inputs/GVL_iXlinker.EtherCAT_Master_EMxxxx.Beckhoff_EM7xxx.A_0005_EM7004_0000_0017.ENC_Inputs_Channel_4.Status/Status_of_input_A <-> ENC Inputs Channel 4/Status/Status of input A
//     PlcTask Inputs/GVL_iXlinker.EtherCAT_Master_EMxxxx.Beckhoff_EM7xxx.A_0005_EM7004_0000_0017.ENC_Inputs_Channel_1.Status/Status_of_input_B <-> ENC Inputs Channel 1/Status/Status of input B
//     PlcTask Inputs/GVL_iXlinker.EtherCAT_Master_EMxxxx.Beckhoff_EM7xxx.A_0005_EM7004_0000_0017.ENC_Inputs_Channel_2.Status/Status_of_input_B <-> ENC Inputs Channel 2/Status/Status of input B
//     PlcTask Inputs/GVL_iXlinker.EtherCAT_Master_EMxxxx.Beckhoff_EM7xxx.A_0005_EM7004_0000_0017.ENC_Inputs_Channel_3.Status/Status_of_input_B <-> ENC Inputs Channel 3/Status/Status of input B
//     PlcTask Inputs/GVL_iXlinker.EtherCAT_Master_EMxxxx.Beckhoff_EM7xxx.A_0005_EM7004_0000_0017.ENC_Inputs_Channel_4.Status/Status_of_input_B <-> ENC Inputs Channel 4/Status/Status of input B
//     PlcTask Inputs/GVL_iXlinker.EtherCAT_Master_EMxxxx.Beckhoff_EM7xxx.A_0005_EM7004_0000_0017.ENC_Inputs_Channel_1.Status/Status_of_input_gate <-> ENC Inputs Channel 1/Status/Status of input gate
//     PlcTask Inputs/GVL_iXlinker.EtherCAT_Master_EMxxxx.Beckhoff_EM7xxx.A_0005_EM7004_0000_0017.ENC_Inputs_Channel_2.Status/Status_of_input_gate <-> ENC Inputs Channel 2/Status/Status of input gate
//     PlcTask Inputs/GVL_iXlinker.EtherCAT_Master_EMxxxx.Beckhoff_EM7xxx.A_0005_EM7004_0000_0017.ENC_Inputs_Channel_3.Status/Status_of_input_gate <-> ENC Inputs Channel 3/Status/Status of input gate
//     PlcTask Inputs/GVL_iXlinker.EtherCAT_Master_EMxxxx.Beckhoff_EM7xxx.A_0005_EM7004_0000_0017.ENC_Inputs_Channel_4.Status/Status_of_input_gate <-> ENC Inputs Channel 4/Status/Status of input gate
//     PlcTask Inputs/GVL_iXlinker.EtherCAT_Master_EMxxxx.Beckhoff_EM7xxx.A_0005_EM7004_0000_0017.ENC_Inputs_Channel_1.Status/Status_of_extern_latch <-> ENC Inputs Channel 1/Status/Status of extern latch
//     PlcTask Inputs/GVL_iXlinker.EtherCAT_Master_EMxxxx.Beckhoff_EM7xxx.A_0005_EM7004_0000_0017.ENC_Inputs_Channel_2.Status/Status_of_extern_latch <-> ENC Inputs Channel 2/Status/Status of extern latch
//     PlcTask Inputs/GVL_iXlinker.EtherCAT_Master_EMxxxx.Beckhoff_EM7xxx.A_0005_EM7004_0000_0017.ENC_Inputs_Channel_3.Status/Status_of_extern_latch <-> ENC Inputs Channel 3/Status/Status of extern latch
//     PlcTask Inputs/GVL_iXlinker.EtherCAT_Master_EMxxxx.Beckhoff_EM7xxx.A_0005_EM7004_0000_0017.ENC_Inputs_Channel_4.Status/Status_of_extern_latch <-> ENC Inputs Channel 4/Status/Status of extern latch
//     PlcTask Inputs/GVL_iXlinker.EtherCAT_Master_EMxxxx.Beckhoff_EM7xxx.A_0005_EM7004_0000_0017.ENC_Inputs_Channel_1.Status/TxPDO_Toggle <-> ENC Inputs Channel 1/Status/TxPDO Toggle
//     PlcTask Inputs/GVL_iXlinker.EtherCAT_Master_EMxxxx.Beckhoff_EM7xxx.A_0005_EM7004_0000_0017.ENC_Inputs_Channel_2.Status/TxPDO_Toggle <-> ENC Inputs Channel 2/Status/TxPDO Toggle
//     PlcTask Inputs/GVL_iXlinker.EtherCAT_Master_EMxxxx.Beckhoff_EM7xxx.A_0005_EM7004_0000_0017.ENC_Inputs_Channel_3.Status/TxPDO_Toggle <-> ENC Inputs Channel 3/Status/TxPDO Toggle
//     PlcTask Inputs/GVL_iXlinker.EtherCAT_Master_EMxxxx.Beckhoff_EM7xxx.A_0005_EM7004_0000_0017.ENC_Inputs_Channel_4.Status/TxPDO_Toggle <-> ENC Inputs Channel 4/Status/TxPDO Toggle
//     PlcTask Inputs/GVL_iXlinker.EtherCAT_Master_EMxxxx.Beckhoff_EM7xxx.A_0005_EM7004_0000_0017.ENC_Inputs_Channel_1.Counter_value <-> ENC Inputs Channel 1/Counter value
//     PlcTask Inputs/GVL_iXlinker.EtherCAT_Master_EMxxxx.Beckhoff_EM7xxx.A_0005_EM7004_0000_0017.ENC_Inputs_Channel_2.Counter_value <-> ENC Inputs Channel 2/Counter value
//     PlcTask Inputs/GVL_iXlinker.EtherCAT_Master_EMxxxx.Beckhoff_EM7xxx.A_0005_EM7004_0000_0017.ENC_Inputs_Channel_3.Counter_value <-> ENC Inputs Channel 3/Counter value
//     PlcTask Inputs/GVL_iXlinker.EtherCAT_Master_EMxxxx.Beckhoff_EM7xxx.A_0005_EM7004_0000_0017.ENC_Inputs_Channel_4.Counter_value <-> ENC Inputs Channel 4/Counter value
//     PlcTask Inputs/GVL_iXlinker.EtherCAT_Master_EMxxxx.Beckhoff_EM7xxx.A_0005_EM7004_0000_0017.ENC_Inputs_Channel_1.Latch_value <-> ENC Inputs Channel 1/Latch value
//     PlcTask Inputs/GVL_iXlinker.EtherCAT_Master_EMxxxx.Beckhoff_EM7xxx.A_0005_EM7004_0000_0017.ENC_Inputs_Channel_2.Latch_value <-> ENC Inputs Channel 2/Latch value
//     PlcTask Inputs/GVL_iXlinker.EtherCAT_Master_EMxxxx.Beckhoff_EM7xxx.A_0005_EM7004_0000_0017.ENC_Inputs_Channel_3.Latch_value <-> ENC Inputs Channel 3/Latch value
//     PlcTask Inputs/GVL_iXlinker.EtherCAT_Master_EMxxxx.Beckhoff_EM7xxx.A_0005_EM7004_0000_0017.ENC_Inputs_Channel_4.Latch_value <-> ENC Inputs Channel 4/Latch value
//     PlcTask Inputs/GVL_iXlinker.EtherCAT_Master_EMxxxx.Beckhoff_EM7xxx.A_0005_EM7004_0000_0017.PLS_Inputs.Status/PLS_Enabled <-> PLS Inputs/Status/PLS Enabled
//     PlcTask Inputs/GVL_iXlinker.EtherCAT_Master_EMxxxx.Beckhoff_EM7xxx.A_0005_EM7004_0000_0017.PLS_Inputs.Status/Unequal_SI_0 <-> PLS Inputs/Status/Unequal SI:0
//     PlcTask Outputs/GVL_iXlinker.EtherCAT_Master_EMxxxx.Beckhoff_EM7xxx.A_0005_EM7004_0000_0017.DO_Outputs.Output/Output_0 <-> DO Outputs/Output/Output 0
//     PlcTask Outputs/GVL_iXlinker.EtherCAT_Master_EMxxxx.Beckhoff_EM7xxx.A_0005_EM7004_0000_0017.DO_Outputs.Output/Output_1 <-> DO Outputs/Output/Output 1
//     PlcTask Outputs/GVL_iXlinker.EtherCAT_Master_EMxxxx.Beckhoff_EM7xxx.A_0005_EM7004_0000_0017.DO_Outputs.Output/Output_2 <-> DO Outputs/Output/Output 2
//     PlcTask Outputs/GVL_iXlinker.EtherCAT_Master_EMxxxx.Beckhoff_EM7xxx.A_0005_EM7004_0000_0017.DO_Outputs.Output/Output_3 <-> DO Outputs/Output/Output 3
//     PlcTask Outputs/GVL_iXlinker.EtherCAT_Master_EMxxxx.Beckhoff_EM7xxx.A_0005_EM7004_0000_0017.DO_Outputs.Output/Output_4 <-> DO Outputs/Output/Output 4
//     PlcTask Outputs/GVL_iXlinker.EtherCAT_Master_EMxxxx.Beckhoff_EM7xxx.A_0005_EM7004_0000_0017.DO_Outputs.Output/Output_5 <-> DO Outputs/Output/Output 5
//     PlcTask Outputs/GVL_iXlinker.EtherCAT_Master_EMxxxx.Beckhoff_EM7xxx.A_0005_EM7004_0000_0017.DO_Outputs.Output/Output_6 <-> DO Outputs/Output/Output 6
//     PlcTask Outputs/GVL_iXlinker.EtherCAT_Master_EMxxxx.Beckhoff_EM7xxx.A_0005_EM7004_0000_0017.DO_Outputs.Output/Output_7 <-> DO Outputs/Output/Output 7
//     PlcTask Outputs/GVL_iXlinker.EtherCAT_Master_EMxxxx.Beckhoff_EM7xxx.A_0005_EM7004_0000_0017.DO_Outputs.Output/Output_8 <-> DO Outputs/Output/Output 8
//     PlcTask Outputs/GVL_iXlinker.EtherCAT_Master_EMxxxx.Beckhoff_EM7xxx.A_0005_EM7004_0000_0017.DO_Outputs.Output/Output_9 <-> DO Outputs/Output/Output 9
//     PlcTask Outputs/GVL_iXlinker.EtherCAT_Master_EMxxxx.Beckhoff_EM7xxx.A_0005_EM7004_0000_0017.DO_Outputs.Output/Output_10 <-> DO Outputs/Output/Output 10
//     PlcTask Outputs/GVL_iXlinker.EtherCAT_Master_EMxxxx.Beckhoff_EM7xxx.A_0005_EM7004_0000_0017.DO_Outputs.Output/Output_11 <-> DO Outputs/Output/Output 11
//     PlcTask Outputs/GVL_iXlinker.EtherCAT_Master_EMxxxx.Beckhoff_EM7xxx.A_0005_EM7004_0000_0017.DO_Outputs.Output/Output_12 <-> DO Outputs/Output/Output 12
//     PlcTask Outputs/GVL_iXlinker.EtherCAT_Master_EMxxxx.Beckhoff_EM7xxx.A_0005_EM7004_0000_0017.DO_Outputs.Output/Output_13 <-> DO Outputs/Output/Output 13
//     PlcTask Outputs/GVL_iXlinker.EtherCAT_Master_EMxxxx.Beckhoff_EM7xxx.A_0005_EM7004_0000_0017.DO_Outputs.Output/Output_14 <-> DO Outputs/Output/Output 14
//     PlcTask Outputs/GVL_iXlinker.EtherCAT_Master_EMxxxx.Beckhoff_EM7xxx.A_0005_EM7004_0000_0017.DO_Outputs.Output/Output_15 <-> DO Outputs/Output/Output 15
//     PlcTask Outputs/GVL_iXlinker.EtherCAT_Master_EMxxxx.Beckhoff_EM7xxx.A_0005_EM7004_0000_0017.AO_Outputs_Channel_1.Analog_output <-> AO Outputs Channel 1/Analog output
//     PlcTask Outputs/GVL_iXlinker.EtherCAT_Master_EMxxxx.Beckhoff_EM7xxx.A_0005_EM7004_0000_0017.AO_Outputs_Channel_2.Analog_output <-> AO Outputs Channel 2/Analog output
//     PlcTask Outputs/GVL_iXlinker.EtherCAT_Master_EMxxxx.Beckhoff_EM7xxx.A_0005_EM7004_0000_0017.AO_Outputs_Channel_3.Analog_output <-> AO Outputs Channel 3/Analog output
//     PlcTask Outputs/GVL_iXlinker.EtherCAT_Master_EMxxxx.Beckhoff_EM7xxx.A_0005_EM7004_0000_0017.AO_Outputs_Channel_4.Analog_output <-> AO Outputs Channel 4/Analog output
//     PlcTask Outputs/GVL_iXlinker.EtherCAT_Master_EMxxxx.Beckhoff_EM7xxx.A_0005_EM7004_0000_0017.ENC_Outputs_Channel_1.Control/Enable_latch_extern_on_positive_edge <-> ENC Outputs Channel 1/Control/Enable latch extern on positive edge
//     PlcTask Outputs/GVL_iXlinker.EtherCAT_Master_EMxxxx.Beckhoff_EM7xxx.A_0005_EM7004_0000_0017.ENC_Outputs_Channel_2.Control/Enable_latch_extern_on_positive_edge <-> ENC Outputs Channel 2/Control/Enable latch extern on positive edge
//     PlcTask Outputs/GVL_iXlinker.EtherCAT_Master_EMxxxx.Beckhoff_EM7xxx.A_0005_EM7004_0000_0017.ENC_Outputs_Channel_3.Control/Enable_latch_extern_on_positive_edge <-> ENC Outputs Channel 3/Control/Enable latch extern on positive edge
//     PlcTask Outputs/GVL_iXlinker.EtherCAT_Master_EMxxxx.Beckhoff_EM7xxx.A_0005_EM7004_0000_0017.ENC_Outputs_Channel_4.Control/Enable_latch_extern_on_positive_edge <-> ENC Outputs Channel 4/Control/Enable latch extern on positive edge
//     PlcTask Outputs/GVL_iXlinker.EtherCAT_Master_EMxxxx.Beckhoff_EM7xxx.A_0005_EM7004_0000_0017.ENC_Outputs_Channel_1.Control/Set_counter <-> ENC Outputs Channel 1/Control/Set counter
//     PlcTask Outputs/GVL_iXlinker.EtherCAT_Master_EMxxxx.Beckhoff_EM7xxx.A_0005_EM7004_0000_0017.ENC_Outputs_Channel_2.Control/Set_counter <-> ENC Outputs Channel 2/Control/Set counter
//     PlcTask Outputs/GVL_iXlinker.EtherCAT_Master_EMxxxx.Beckhoff_EM7xxx.A_0005_EM7004_0000_0017.ENC_Outputs_Channel_3.Control/Set_counter <-> ENC Outputs Channel 3/Control/Set counter
//     PlcTask Outputs/GVL_iXlinker.EtherCAT_Master_EMxxxx.Beckhoff_EM7xxx.A_0005_EM7004_0000_0017.ENC_Outputs_Channel_4.Control/Set_counter <-> ENC Outputs Channel 4/Control/Set counter
//     PlcTask Outputs/GVL_iXlinker.EtherCAT_Master_EMxxxx.Beckhoff_EM7xxx.A_0005_EM7004_0000_0017.ENC_Outputs_Channel_1.Control/Enable_latch_extern_on_negative_edge <-> ENC Outputs Channel 1/Control/Enable latch extern on negative edge
//     PlcTask Outputs/GVL_iXlinker.EtherCAT_Master_EMxxxx.Beckhoff_EM7xxx.A_0005_EM7004_0000_0017.ENC_Outputs_Channel_2.Control/Enable_latch_extern_on_negative_edge <-> ENC Outputs Channel 2/Control/Enable latch extern on negative edge
//     PlcTask Outputs/GVL_iXlinker.EtherCAT_Master_EMxxxx.Beckhoff_EM7xxx.A_0005_EM7004_0000_0017.ENC_Outputs_Channel_3.Control/Enable_latch_extern_on_negative_edge <-> ENC Outputs Channel 3/Control/Enable latch extern on negative edge
//     PlcTask Outputs/GVL_iXlinker.EtherCAT_Master_EMxxxx.Beckhoff_EM7xxx.A_0005_EM7004_0000_0017.ENC_Outputs_Channel_4.Control/Enable_latch_extern_on_negative_edge <-> ENC Outputs Channel 4/Control/Enable latch extern on negative edge
//     PlcTask Outputs/GVL_iXlinker.EtherCAT_Master_EMxxxx.Beckhoff_EM7xxx.A_0005_EM7004_0000_0017.ENC_Outputs_Channel_1.Set_counter_value <-> ENC Outputs Channel 1/Set counter value
//     PlcTask Outputs/GVL_iXlinker.EtherCAT_Master_EMxxxx.Beckhoff_EM7xxx.A_0005_EM7004_0000_0017.ENC_Outputs_Channel_2.Set_counter_value <-> ENC Outputs Channel 2/Set counter value
//     PlcTask Outputs/GVL_iXlinker.EtherCAT_Master_EMxxxx.Beckhoff_EM7xxx.A_0005_EM7004_0000_0017.ENC_Outputs_Channel_3.Set_counter_value <-> ENC Outputs Channel 3/Set counter value
//     PlcTask Outputs/GVL_iXlinker.EtherCAT_Master_EMxxxx.Beckhoff_EM7xxx.A_0005_EM7004_0000_0017.ENC_Outputs_Channel_4.Set_counter_value <-> ENC Outputs Channel 4/Set counter value
//     PlcTask Outputs/GVL_iXlinker.EtherCAT_Master_EMxxxx.Beckhoff_EM7xxx.A_0005_EM7004_0000_0017.PLS_Outputs.Control/Enable_PLS <-> PLS Outputs/Control/Enable PLS
//     PlcTask Inputs/GVL_iXlinker.EtherCAT_Master_EMxxxx.Beckhoff_EM7xxx.A_0005_EM7004_0000_0017.WcState.WcState <-> WcState/WcState
//     PlcTask Inputs/GVL_iXlinker.EtherCAT_Master_EMxxxx.Beckhoff_EM7xxx.A_0005_EM7004_0000_0017.WcState.InputToggle <-> WcState/InputToggle
//     PlcTask Inputs/GVL_iXlinker.EtherCAT_Master_EMxxxx.Beckhoff_EM7xxx.A_0005_EM7004_0000_0017.InfoData.AdsAddr <-> InfoData/AdsAddr
//     PlcTask Inputs/GVL_iXlinker.EtherCAT_Master_EMxxxx.Beckhoff_EM7xxx.A_0005_EM7004_0000_0017.InfoData.State <-> InfoData/State
//   PLC/PLC Instance <-> EtherCAT Master EMxxxx/Beckhoff EM7xxx/A_0006(EM7004-0000-0018)
//     PlcTask Inputs/GVL_iXlinker.EtherCAT_Master_EMxxxx.Beckhoff_EM7xxx.A_0006_EM7004_0000_0018.DI_Inputs.Input/Input_0 <-> DI Inputs/Input/Input 0
//     PlcTask Inputs/GVL_iXlinker.EtherCAT_Master_EMxxxx.Beckhoff_EM7xxx.A_0006_EM7004_0000_0018.DI_Inputs.Input/Input_1 <-> DI Inputs/Input/Input 1
//     PlcTask Inputs/GVL_iXlinker.EtherCAT_Master_EMxxxx.Beckhoff_EM7xxx.A_0006_EM7004_0000_0018.DI_Inputs.Input/Input_2 <-> DI Inputs/Input/Input 2
//     PlcTask Inputs/GVL_iXlinker.EtherCAT_Master_EMxxxx.Beckhoff_EM7xxx.A_0006_EM7004_0000_0018.DI_Inputs.Input/Input_3 <-> DI Inputs/Input/Input 3
//     PlcTask Inputs/GVL_iXlinker.EtherCAT_Master_EMxxxx.Beckhoff_EM7xxx.A_0006_EM7004_0000_0018.DI_Inputs.Input/Input_4 <-> DI Inputs/Input/Input 4
//     PlcTask Inputs/GVL_iXlinker.EtherCAT_Master_EMxxxx.Beckhoff_EM7xxx.A_0006_EM7004_0000_0018.DI_Inputs.Input/Input_5 <-> DI Inputs/Input/Input 5
//     PlcTask Inputs/GVL_iXlinker.EtherCAT_Master_EMxxxx.Beckhoff_EM7xxx.A_0006_EM7004_0000_0018.DI_Inputs.Input/Input_6 <-> DI Inputs/Input/Input 6
//     PlcTask Inputs/GVL_iXlinker.EtherCAT_Master_EMxxxx.Beckhoff_EM7xxx.A_0006_EM7004_0000_0018.DI_Inputs.Input/Input_7 <-> DI Inputs/Input/Input 7
//     PlcTask Inputs/GVL_iXlinker.EtherCAT_Master_EMxxxx.Beckhoff_EM7xxx.A_0006_EM7004_0000_0018.DI_Inputs.Input/Input_8 <-> DI Inputs/Input/Input 8
//     PlcTask Inputs/GVL_iXlinker.EtherCAT_Master_EMxxxx.Beckhoff_EM7xxx.A_0006_EM7004_0000_0018.DI_Inputs.Input/Input_9 <-> DI Inputs/Input/Input 9
//     PlcTask Inputs/GVL_iXlinker.EtherCAT_Master_EMxxxx.Beckhoff_EM7xxx.A_0006_EM7004_0000_0018.DI_Inputs.Input/Input_10 <-> DI Inputs/Input/Input 10
//     PlcTask Inputs/GVL_iXlinker.EtherCAT_Master_EMxxxx.Beckhoff_EM7xxx.A_0006_EM7004_0000_0018.DI_Inputs.Input/Input_11 <-> DI Inputs/Input/Input 11
//     PlcTask Inputs/GVL_iXlinker.EtherCAT_Master_EMxxxx.Beckhoff_EM7xxx.A_0006_EM7004_0000_0018.DI_Inputs.Input/Input_12 <-> DI Inputs/Input/Input 12
//     PlcTask Inputs/GVL_iXlinker.EtherCAT_Master_EMxxxx.Beckhoff_EM7xxx.A_0006_EM7004_0000_0018.DI_Inputs.Input/Input_13 <-> DI Inputs/Input/Input 13
//     PlcTask Inputs/GVL_iXlinker.EtherCAT_Master_EMxxxx.Beckhoff_EM7xxx.A_0006_EM7004_0000_0018.DI_Inputs.Input/Input_14 <-> DI Inputs/Input/Input 14
//     PlcTask Inputs/GVL_iXlinker.EtherCAT_Master_EMxxxx.Beckhoff_EM7xxx.A_0006_EM7004_0000_0018.DI_Inputs.Input/Input_15 <-> DI Inputs/Input/Input 15
//     PlcTask Inputs/GVL_iXlinker.EtherCAT_Master_EMxxxx.Beckhoff_EM7xxx.A_0006_EM7004_0000_0018.ENC_Inputs_Channel_1.Status/Latch_extern_valid <-> ENC Inputs Channel 1/Status/Latch extern valid
//     PlcTask Inputs/GVL_iXlinker.EtherCAT_Master_EMxxxx.Beckhoff_EM7xxx.A_0006_EM7004_0000_0018.ENC_Inputs_Channel_2.Status/Latch_extern_valid <-> ENC Inputs Channel 2/Status/Latch extern valid
//     PlcTask Inputs/GVL_iXlinker.EtherCAT_Master_EMxxxx.Beckhoff_EM7xxx.A_0006_EM7004_0000_0018.ENC_Inputs_Channel_3.Status/Latch_extern_valid <-> ENC Inputs Channel 3/Status/Latch extern valid
//     PlcTask Inputs/GVL_iXlinker.EtherCAT_Master_EMxxxx.Beckhoff_EM7xxx.A_0006_EM7004_0000_0018.ENC_Inputs_Channel_4.Status/Latch_extern_valid <-> ENC Inputs Channel 4/Status/Latch extern valid
//     PlcTask Inputs/GVL_iXlinker.EtherCAT_Master_EMxxxx.Beckhoff_EM7xxx.A_0006_EM7004_0000_0018.ENC_Inputs_Channel_1.Status/Set_counter_done <-> ENC Inputs Channel 1/Status/Set counter done
//     PlcTask Inputs/GVL_iXlinker.EtherCAT_Master_EMxxxx.Beckhoff_EM7xxx.A_0006_EM7004_0000_0018.ENC_Inputs_Channel_2.Status/Set_counter_done <-> ENC Inputs Channel 2/Status/Set counter done
//     PlcTask Inputs/GVL_iXlinker.EtherCAT_Master_EMxxxx.Beckhoff_EM7xxx.A_0006_EM7004_0000_0018.ENC_Inputs_Channel_3.Status/Set_counter_done <-> ENC Inputs Channel 3/Status/Set counter done
//     PlcTask Inputs/GVL_iXlinker.EtherCAT_Master_EMxxxx.Beckhoff_EM7xxx.A_0006_EM7004_0000_0018.ENC_Inputs_Channel_4.Status/Set_counter_done <-> ENC Inputs Channel 4/Status/Set counter done
//     PlcTask Inputs/GVL_iXlinker.EtherCAT_Master_EMxxxx.Beckhoff_EM7xxx.A_0006_EM7004_0000_0018.ENC_Inputs_Channel_1.Status/Status_of_input_A <-> ENC Inputs Channel 1/Status/Status of input A
//     PlcTask Inputs/GVL_iXlinker.EtherCAT_Master_EMxxxx.Beckhoff_EM7xxx.A_0006_EM7004_0000_0018.ENC_Inputs_Channel_2.Status/Status_of_input_A <-> ENC Inputs Channel 2/Status/Status of input A
//     PlcTask Inputs/GVL_iXlinker.EtherCAT_Master_EMxxxx.Beckhoff_EM7xxx.A_0006_EM7004_0000_0018.ENC_Inputs_Channel_3.Status/Status_of_input_A <-> ENC Inputs Channel 3/Status/Status of input A
//     PlcTask Inputs/GVL_iXlinker.EtherCAT_Master_EMxxxx.Beckhoff_EM7xxx.A_0006_EM7004_0000_0018.ENC_Inputs_Channel_4.Status/Status_of_input_A <-> ENC Inputs Channel 4/Status/Status of input A
//     PlcTask Inputs/GVL_iXlinker.EtherCAT_Master_EMxxxx.Beckhoff_EM7xxx.A_0006_EM7004_0000_0018.ENC_Inputs_Channel_1.Status/Status_of_input_B <-> ENC Inputs Channel 1/Status/Status of input B
//     PlcTask Inputs/GVL_iXlinker.EtherCAT_Master_EMxxxx.Beckhoff_EM7xxx.A_0006_EM7004_0000_0018.ENC_Inputs_Channel_2.Status/Status_of_input_B <-> ENC Inputs Channel 2/Status/Status of input B
//     PlcTask Inputs/GVL_iXlinker.EtherCAT_Master_EMxxxx.Beckhoff_EM7xxx.A_0006_EM7004_0000_0018.ENC_Inputs_Channel_3.Status/Status_of_input_B <-> ENC Inputs Channel 3/Status/Status of input B
//     PlcTask Inputs/GVL_iXlinker.EtherCAT_Master_EMxxxx.Beckhoff_EM7xxx.A_0006_EM7004_0000_0018.ENC_Inputs_Channel_4.Status/Status_of_input_B <-> ENC Inputs Channel 4/Status/Status of input B
//     PlcTask Inputs/GVL_iXlinker.EtherCAT_Master_EMxxxx.Beckhoff_EM7xxx.A_0006_EM7004_0000_0018.ENC_Inputs_Channel_1.Status/Status_of_input_gate <-> ENC Inputs Channel 1/Status/Status of input gate
//     PlcTask Inputs/GVL_iXlinker.EtherCAT_Master_EMxxxx.Beckhoff_EM7xxx.A_0006_EM7004_0000_0018.ENC_Inputs_Channel_2.Status/Status_of_input_gate <-> ENC Inputs Channel 2/Status/Status of input gate
//     PlcTask Inputs/GVL_iXlinker.EtherCAT_Master_EMxxxx.Beckhoff_EM7xxx.A_0006_EM7004_0000_0018.ENC_Inputs_Channel_3.Status/Status_of_input_gate <-> ENC Inputs Channel 3/Status/Status of input gate
//     PlcTask Inputs/GVL_iXlinker.EtherCAT_Master_EMxxxx.Beckhoff_EM7xxx.A_0006_EM7004_0000_0018.ENC_Inputs_Channel_4.Status/Status_of_input_gate <-> ENC Inputs Channel 4/Status/Status of input gate
//     PlcTask Inputs/GVL_iXlinker.EtherCAT_Master_EMxxxx.Beckhoff_EM7xxx.A_0006_EM7004_0000_0018.ENC_Inputs_Channel_1.Status/Status_of_extern_latch <-> ENC Inputs Channel 1/Status/Status of extern latch
//     PlcTask Inputs/GVL_iXlinker.EtherCAT_Master_EMxxxx.Beckhoff_EM7xxx.A_0006_EM7004_0000_0018.ENC_Inputs_Channel_2.Status/Status_of_extern_latch <-> ENC Inputs Channel 2/Status/Status of extern latch
//     PlcTask Inputs/GVL_iXlinker.EtherCAT_Master_EMxxxx.Beckhoff_EM7xxx.A_0006_EM7004_0000_0018.ENC_Inputs_Channel_3.Status/Status_of_extern_latch <-> ENC Inputs Channel 3/Status/Status of extern latch
//     PlcTask Inputs/GVL_iXlinker.EtherCAT_Master_EMxxxx.Beckhoff_EM7xxx.A_0006_EM7004_0000_0018.ENC_Inputs_Channel_4.Status/Status_of_extern_latch <-> ENC Inputs Channel 4/Status/Status of extern latch
//     PlcTask Inputs/GVL_iXlinker.EtherCAT_Master_EMxxxx.Beckhoff_EM7xxx.A_0006_EM7004_0000_0018.ENC_Inputs_Channel_1.Status/TxPDO_Toggle <-> ENC Inputs Channel 1/Status/TxPDO Toggle
//     PlcTask Inputs/GVL_iXlinker.EtherCAT_Master_EMxxxx.Beckhoff_EM7xxx.A_0006_EM7004_0000_0018.ENC_Inputs_Channel_2.Status/TxPDO_Toggle <-> ENC Inputs Channel 2/Status/TxPDO Toggle
//     PlcTask Inputs/GVL_iXlinker.EtherCAT_Master_EMxxxx.Beckhoff_EM7xxx.A_0006_EM7004_0000_0018.ENC_Inputs_Channel_3.Status/TxPDO_Toggle <-> ENC Inputs Channel 3/Status/TxPDO Toggle
//     PlcTask Inputs/GVL_iXlinker.EtherCAT_Master_EMxxxx.Beckhoff_EM7xxx.A_0006_EM7004_0000_0018.ENC_Inputs_Channel_4.Status/TxPDO_Toggle <-> ENC Inputs Channel 4/Status/TxPDO Toggle
//     PlcTask Inputs/GVL_iXlinker.EtherCAT_Master_EMxxxx.Beckhoff_EM7xxx.A_0006_EM7004_0000_0018.ENC_Inputs_Channel_1.Counter_value <-> ENC Inputs Channel 1/Counter value
//     PlcTask Inputs/GVL_iXlinker.EtherCAT_Master_EMxxxx.Beckhoff_EM7xxx.A_0006_EM7004_0000_0018.ENC_Inputs_Channel_2.Counter_value <-> ENC Inputs Channel 2/Counter value
//     PlcTask Inputs/GVL_iXlinker.EtherCAT_Master_EMxxxx.Beckhoff_EM7xxx.A_0006_EM7004_0000_0018.ENC_Inputs_Channel_3.Counter_value <-> ENC Inputs Channel 3/Counter value
//     PlcTask Inputs/GVL_iXlinker.EtherCAT_Master_EMxxxx.Beckhoff_EM7xxx.A_0006_EM7004_0000_0018.ENC_Inputs_Channel_4.Counter_value <-> ENC Inputs Channel 4/Counter value
//     PlcTask Inputs/GVL_iXlinker.EtherCAT_Master_EMxxxx.Beckhoff_EM7xxx.A_0006_EM7004_0000_0018.ENC_Inputs_Channel_1.Latch_value <-> ENC Inputs Channel 1/Latch value
//     PlcTask Inputs/GVL_iXlinker.EtherCAT_Master_EMxxxx.Beckhoff_EM7xxx.A_0006_EM7004_0000_0018.ENC_Inputs_Channel_2.Latch_value <-> ENC Inputs Channel 2/Latch value
